LIN {X 0,Y 466.708,Z 598.278,A -85,B 0,C 180,E1 -7470,E2 -7470} C_VEL
LIN {X 0,Y 466.926,Z 594.295,A -85,B 0,C 180,E1 -7471.294,E2 -7471.294} C_VEL
LIN {X 0,Y 467.015,Z 589.345,A -85,B 0,C 180,E1 -7472.587,E2 -7472.587} C_VEL
LIN {X 0,Y 467.543,Z 582.26,A -85,B 0,C 180,E1 -7474.094,E2 -7474.094} C_VEL
LIN {X 0,Y 468.033,Z 573.535,A -85,B 0,C 180,E1 -7475.601,E2 -7475.601} C_VEL
LIN {X 0,Y 468.642,Z 564.398,A -85,B 0,C 180,E1 -7476.89,E2 -7476.89} C_VEL
LIN {X 0,Y 469.162,Z 555.335,A -85,B 0,C 180,E1 -7477.96,E2 -7477.96} C_VEL
LIN {X 0,Y 469.742,Z 543.987,A -85,B 0,C 180,E1 -7479.082,E2 -7479.082} C_VEL
LIN {X 0,Y 470.435,Z 532.566,A -85,B 0,C 180,E1 -7480.001,E2 -7480.001} C_VEL
LIN {X 0,Y 471.079,Z 519.327,A -85,B 0,C 180,E1 -7480.856,E2 -7480.856} C_VEL
LIN {X 0,Y 471.604,Z 506.561,A -85,B 0,C 180,E1 -7481.497,E2 -7481.497} C_VEL
LIN {X 0,Y 472.126,Z 492.888,A -85,B 0,C 180,E1 -7482.001,E2 -7482.001} C_VEL
LIN {X 0,Y 472.334,Z 478.929,A -85,B 0,C 180,E1 -7482.35,E2 -7482.35} C_VEL
LIN {X 0,Y 473.44,Z 363.18,A -85,B 0,C 180,E1 -7484.133,E2 -7484.133} C_VEL
LIN {X 0,Y 469.666,Z 345.085,A -85,B 0,C 180,E1 -7484.585,E2 -7484.585} C_VEL
LIN {X 0,Y 469.849,Z 337.166,A -85,B 0,C 180,E1 -7486.064,E2 -7486.064} C_VEL
LIN {X 0,Y 467.678,Z 325.858,A -85,B 0,C 180,E1 -7488.367,E2 -7488.367} C_VEL
LIN {X 0,Y 467.584,Z 325.868,A -85,B 0,C 180,E1 -7491.267,E2 -7491.267} C_VEL
LIN {X 0,Y 467.566,Z 325.871,A -85,B 0,C 180,E1 -7493.943,E2 -7493.943} C_VEL
LIN {X 0,Y 467.615,Z 325.859,A -85,B 0,C 180,E1 -7496.8,E2 -7496.8} C_VEL
LIN {X 0,Y 467.555,Z 325.871,A -85,B 0,C 180,E1 -7499.737,E2 -7499.737} C_VEL
LIN {X 0,Y 467.584,Z 325.862,A -85,B 0,C 180,E1 -7502.757,E2 -7502.757} C_VEL
LIN {X 0,Y 467.556,Z 325.867,A -85,B 0,C 180,E1 -7505.888,E2 -7505.888} C_VEL
LIN {X 0,Y 467.581,Z 325.865,A -85,B 0,C 180,E1 -7509.144,E2 -7509.144} C_VEL
LIN {X 0,Y 467.584,Z 325.861,A -85,B 0,C 180,E1 -7512.566,E2 -7512.566} C_VEL
LIN {X 0,Y 467.567,Z 325.866,A -85,B 0,C 180,E1 -7515.052,E2 -7515.052} C_VEL
LIN {X 0,Y 467.585,Z 325.866,A -85,B 0,C 180,E1 -7517.439,E2 -7517.439} C_VEL
LIN {X 0,Y 467.57,Z 325.866,A -85,B 0,C 180,E1 -7520.853,E2 -7520.853} C_VEL
LIN {X 0,Y 467.552,Z 325.866,A -85,B 0,C 180,E1 -7524.26,E2 -7524.26} C_VEL
LIN {X 0,Y 467.572,Z 325.868,A -85,B 0,C 180,E1 -7527.32,E2 -7527.32} C_VEL
LIN {X 0,Y 467.56,Z 325.867,A -85,B 0,C 180,E1 -7530.667,E2 -7530.667} C_VEL
LIN {X 0,Y 467.578,Z 325.863,A -85,B 0,C 180,E1 -7533.197,E2 -7533.197} C_VEL
LIN {X 0,Y 467.579,Z 325.864,A -85,B 0,C 180,E1 -7536.468,E2 -7536.468} C_VEL
LIN {X 0,Y 467.61,Z 325.85,A -85,B 0,C 180,E1 -7539.776,E2 -7539.776} C_VEL
LIN {X 0,Y 467.583,Z 325.863,A -85,B 0,C 180,E1 -7542.505,E2 -7542.505} C_VEL
LIN {X 0,Y 467.589,Z 325.86,A -85,B 0,C 180,E1 -7545.196,E2 -7545.196} C_VEL
LIN {X 0,Y 467.643,Z 325.845,A -85,B 0,C 180,E1 -7547.854,E2 -7547.854} C_VEL
LIN {X 0,Y 467.654,Z 325.854,A -85,B 0,C 180,E1 -7551.356,E2 -7551.356} C_VEL
LIN {X 0,Y 467.71,Z 325.843,A -85,B 0,C 180,E1 -7553.962,E2 -7553.962} C_VEL
LIN {X 0,Y 467.808,Z 325.831,A -85,B 0,C 180,E1 -7557.417,E2 -7557.417} C_VEL
LIN {X 0,Y 467.832,Z 325.832,A -85,B 0,C 180,E1 -7560,E2 -7560} C_VEL
LIN {X 0,Y 467.796,Z 325.835,A -85,B 0,C 180,E1 -7562.583,E2 -7562.583} C_VEL
LIN {X 0,Y 467.69,Z 325.851,A -85,B 0,C 180,E1 -7566.038,E2 -7566.038} C_VEL
LIN {X 0,Y 467.642,Z 325.853,A -85,B 0,C 180,E1 -7568.643,E2 -7568.643} C_VEL
LIN {X 0,Y 467.642,Z 325.859,A -85,B 0,C 180,E1 -7572.146,E2 -7572.146} C_VEL
LIN {X 0,Y 467.625,Z 325.853,A -85,B 0,C 180,E1 -7575.695,E2 -7575.695} C_VEL
LIN {X 0,Y 467.608,Z 325.858,A -85,B 0,C 180,E1 -7579.308,E2 -7579.308} C_VEL
LIN {X 0,Y 467.522,Z 325.87,A -85,B 0,C 180,E1 -7582.074,E2 -7582.074} C_VEL
LIN {X 0,Y 467.571,Z 325.861,A -85,B 0,C 180,E1 -7584.889,E2 -7584.889} C_VEL
LIN {X 0,Y 467.569,Z 325.866,A -85,B 0,C 180,E1 -7587.772,E2 -7587.772} C_VEL
LIN {X 0,Y 467.557,Z 325.863,A -85,B 0,C 180,E1 -7591.045,E2 -7591.045} C_VEL
LIN {X 0,Y 467.579,Z 325.865,A -85,B 0,C 180,E1 -7594.243,E2 -7594.243} C_VEL
LIN {X 0,Y 467.54,Z 325.868,A -85,B 0,C 180,E1 -7597.187,E2 -7597.187} C_VEL
LIN {X 0,Y 467.569,Z 325.862,A -85,B 0,C 180,E1 -7600.265,E2 -7600.265} C_VEL
LIN {X 0,Y 467.579,Z 325.861,A -85,B 0,C 180,E1 -7602.568,E2 -7602.568} C_VEL
LIN {X 0,Y 467.563,Z 325.865,A -85,B 0,C 180,E1 -7605.054,E2 -7605.054} C_VEL
LIN {X 0,Y 467.583,Z 325.867,A -85,B 0,C 180,E1 -7607.441,E2 -7607.441} C_VEL
LIN {X 0,Y 467.555,Z 325.869,A -85,B 0,C 180,E1 -7610.854,E2 -7610.854} C_VEL
LIN {X 0,Y 467.558,Z 325.869,A -85,B 0,C 180,E1 -7614.261,E2 -7614.261} C_VEL
LIN {X 0,Y 467.578,Z 325.87,A -85,B 0,C 180,E1 -7617.322,E2 -7617.322} C_VEL
LIN {X 0,Y 467.567,Z 325.867,A -85,B 0,C 180,E1 -7620.668,E2 -7620.668} C_VEL
LIN {X 0,Y 467.633,Z 325.91,A -85,B 0,C 180,E1 -7622.233,E2 -7622.233} C_VEL
LIN {X 0,Y 470.717,Z 340.455,A -85,B 0,C 180,E1 -7624.817,E2 -7624.817} C_VEL
LIN {X 0,Y 470.568,Z 347.177,A -85,B 0,C 180,E1 -7625.912,E2 -7625.912} C_VEL
LIN {X 0,Y 469.722,Z 364.766,A -85,B 0,C 180,E1 -7628.727,E2 -7628.727} C_VEL
LIN {X 0,Y 469.505,Z 369.198,A -85,B 0,C 180,E1 -7629.43,E2 -7629.43} C_VEL
LIN {X 0,Y 473.306,Z 391.122,A -85,B 0,C 180,E1 -7629.942,E2 -7629.942} C_VEL
LIN {X 0,Y 472.118,Z 506.928,A -85,B 0,C 180,E1 -7631.728,E2 -7631.728} C_VEL
LIN {X 0,Y 471.704,Z 521.762,A -85,B 0,C 180,E1 -7632.133,E2 -7632.133} C_VEL
LIN {X 0,Y 471.22,Z 535.785,A -85,B 0,C 180,E1 -7632.699,E2 -7632.699} C_VEL
LIN {X 0,Y 470.593,Z 549.174,A -85,B 0,C 180,E1 -7633.423,E2 -7633.423} C_VEL
LIN {X 0,Y 469.936,Z 561.542,A -85,B 0,C 180,E1 -7634.273,E2 -7634.273} C_VEL
LIN {X 0,Y 469.206,Z 573.078,A -85,B 0,C 180,E1 -7635.249,E2 -7635.249} C_VEL
LIN {X 0,Y 468.599,Z 583.669,A -85,B 0,C 180,E1 -7636.337,E2 -7636.337} C_VEL
LIN {X 0,Y 468.155,Z 593.288,A -85,B 0,C 180,E1 -7637.527,E2 -7637.527} C_VEL
LIN {X 0,Y 467.605,Z 602.864,A -85,B 0,C 180,E1 -7638.952,E2 -7638.952} C_VEL
LIN {X 0,Y 467.212,Z 611.173,A -85,B 0,C 180,E1 -7640.476,E2 -7640.476} C_VEL
LIN {X 0,Y 466.95,Z 616.974,A -85,B 0,C 180,E1 -7641.78,E2 -7641.78} C_VEL
LIN {X 0,Y 466.824,Z 621.733,A -85,B 0,C 180,E1 -7643.083,E2 -7643.083} C_VEL
LIN {X 0,Y 466.73,Z 626.661,A -85,B 0,C 180,E1 -7644.817,E2 -7644.817} C_VEL
LIN {X 0,Y 466.679,Z 630.086,A -85,B 0,C 180,E1 -7646.547,E2 -7646.547} C_VEL
LIN {X 0,Y 466.604,Z 632.111,A -85,B 0,C 180,E1 -7648.274,E2 -7648.274} C_VEL
LIN {X 0,Y 466.597,Z 632.785,A -85,B 0,C 180,E1 -7650,E2 -7650} C_VEL
LIN {X 0,Y 466.604,Z 632.119,A -85,B 0,C 180,E1 -7651.726,E2 -7651.726} C_VEL
LIN {X 0,Y 466.679,Z 630.104,A -85,B 0,C 180,E1 -7653.453,E2 -7653.453} C_VEL
LIN {X 0,Y 466.731,Z 626.692,A -85,B 0,C 180,E1 -7655.183,E2 -7655.183} C_VEL
LIN {X 0,Y 466.82,Z 621.782,A -85,B 0,C 180,E1 -7656.917,E2 -7656.917} C_VEL
LIN {X 0,Y 467.036,Z 615.237,A -85,B 0,C 180,E1 -7658.655,E2 -7658.655} C_VEL
LIN {X 0,Y 467.312,Z 607.962,A -85,B 0,C 180,E1 -7660.178,E2 -7660.178} C_VEL
LIN {X 0,Y 467.865,Z 598.973,A -85,B 0,C 180,E1 -7661.7,E2 -7661.7} C_VEL
LIN {X 0,Y 468.351,Z 589.551,A -85,B 0,C 180,E1 -7663.008,E2 -7663.008} C_VEL
LIN {X 0,Y 468.939,Z 579.134,A -85,B 0,C 180,E1 -7664.206,E2 -7664.206} C_VEL
LIN {X 0,Y 469.638,Z 567.661,A -85,B 0,C 180,E1 -7665.292,E2 -7665.292} C_VEL
LIN {X 0,Y 470.388,Z 554.968,A -85,B 0,C 180,E1 -7666.268,E2 -7666.268} C_VEL
LIN {X 0,Y 471.078,Z 542.255,A -85,B 0,C 180,E1 -7667.045,E2 -7667.045} C_VEL
LIN {X 0,Y 471.591,Z 528.59,A -85,B 0,C 180,E1 -7667.693,E2 -7667.693} C_VEL
LIN {X 0,Y 472.162,Z 513.986,A -85,B 0,C 180,E1 -7668.183,E2 -7668.183} C_VEL
LIN {X 0,Y 472.475,Z 499.718,A -85,B 0,C 180,E1 -7668.482,E2 -7668.482} C_VEL
LIN {X 0,Y 473.547,Z 391.005,A -85,B 0,C 180,E1 -7670.161,E2 -7670.161} C_VEL
LIN {X 0,Y 470.028,Z 371.07,A -85,B 0,C 180,E1 -7670.65,E2 -7670.65} C_VEL
LIN {X 0,Y 469.681,Z 368.925,A -85,B 0,C 180,E1 -7670.736,E2 -7670.736} C_VEL
LIN {X 0,Y 470.564,Z 351.6,A -85,B 0,C 180,E1 -7673.547,E2 -7673.547} C_VEL
LIN {X 0,Y 471.044,Z 341.783,A -85,B 0,C 180,E1 -7675.164,E2 -7675.164} C_VEL
LIN {X 0,Y 468.173,Z 328.175,A -85,B 0,C 180,E1 -7677.665,E2 -7677.665} C_VEL
LIN {X 0,Y 467.608,Z 325.863,A -85,B 0,C 180,E1 -7678.134,E2 -7678.134} C_VEL
LIN {X 0,Y 467.579,Z 325.867,A -85,B 0,C 180,E1 -7681.739,E2 -7681.739} C_VEL
LIN {X 0,Y 467.564,Z 325.868,A -85,B 0,C 180,E1 -7684.832,E2 -7684.832} C_VEL
LIN {X 0,Y 467.561,Z 325.862,A -85,B 0,C 180,E1 -7688.044,E2 -7688.044} C_VEL
LIN {X 0,Y 467.572,Z 325.859,A -85,B 0,C 180,E1 -7691.276,E2 -7691.276} C_VEL
LIN {X 0,Y 467.544,Z 325.866,A -85,B 0,C 180,E1 -7693.82,E2 -7693.82} C_VEL
LIN {X 0,Y 467.549,Z 325.871,A -85,B 0,C 180,E1 -7696.255,E2 -7696.255} C_VEL
LIN {X 0,Y 467.57,Z 325.865,A -85,B 0,C 180,E1 -7698.722,E2 -7698.722} C_VEL
LIN {X 0,Y 467.557,Z 325.872,A -85,B 0,C 180,E1 -7701.955,E2 -7701.955} C_VEL
LIN {X 0,Y 467.557,Z 325.863,A -85,B 0,C 180,E1 -7705.167,E2 -7705.167} C_VEL
LIN {X 0,Y 467.572,Z 325.861,A -85,B 0,C 180,E1 -7708.259,E2 -7708.259} C_VEL
LIN {X 0,Y 467.544,Z 325.859,A -85,B 0,C 180,E1 -7711.248,E2 -7711.248} C_VEL
LIN {X 0,Y 467.572,Z 325.866,A -85,B 0,C 180,E1 -7714.158,E2 -7714.158} C_VEL
LIN {X 0,Y 467.564,Z 325.864,A -85,B 0,C 180,E1 -7716.995,E2 -7716.995} C_VEL
LIN {X 0,Y 467.609,Z 325.861,A -85,B 0,C 180,E1 -7719.777,E2 -7719.777} C_VEL
LIN {X 0,Y 467.581,Z 325.862,A -85,B 0,C 180,E1 -7722.506,E2 -7722.506} C_VEL
LIN {X 0,Y 467.586,Z 325.862,A -85,B 0,C 180,E1 -7725.196,E2 -7725.196} C_VEL
LIN {X 0,Y 467.633,Z 325.856,A -85,B 0,C 180,E1 -7727.854,E2 -7727.854} C_VEL
LIN {X 0,Y 467.615,Z 325.864,A -85,B 0,C 180,E1 -7731.356,E2 -7731.356} C_VEL
LIN {X 0,Y 467.695,Z 325.85,A -85,B 0,C 180,E1 -7733.962,E2 -7733.962} C_VEL
LIN {X 0,Y 467.804,Z 325.836,A -85,B 0,C 180,E1 -7737.417,E2 -7737.417} C_VEL
LIN {X 0,Y 467.833,Z 325.832,A -85,B 0,C 180,E1 -7740,E2 -7740} C_VEL
LIN {X 0,Y 467.834,Z 325.827,A -85,B 0,C 180,E1 -7742.583,E2 -7742.583} C_VEL
LIN {X 0,Y 467.711,Z 325.845,A -85,B 0,C 180,E1 -7746.038,E2 -7746.038} C_VEL
LIN {X 0,Y 467.655,Z 325.852,A -85,B 0,C 180,E1 -7748.644,E2 -7748.644} C_VEL
LIN {X 0,Y 467.643,Z 325.849,A -85,B 0,C 180,E1 -7752.146,E2 -7752.146} C_VEL
LIN {X 0,Y 467.627,Z 325.855,A -85,B 0,C 180,E1 -7755.696,E2 -7755.696} C_VEL
LIN {X 0,Y 467.611,Z 325.861,A -85,B 0,C 180,E1 -7759.309,E2 -7759.309} C_VEL
LIN {X 0,Y 467.524,Z 325.869,A -85,B 0,C 180,E1 -7762.075,E2 -7762.075} C_VEL
LIN {X 0,Y 467.593,Z 325.864,A -85,B 0,C 180,E1 -7764.888,E2 -7764.888} C_VEL
LIN {X 0,Y 467.611,Z 325.856,A -85,B 0,C 180,E1 -7767.77,E2 -7767.77} C_VEL
LIN {X 0,Y 467.561,Z 325.866,A -85,B 0,C 180,E1 -7771.046,E2 -7771.046} C_VEL
LIN {X 0,Y 467.582,Z 325.864,A -85,B 0,C 180,E1 -7774.243,E2 -7774.243} C_VEL
LIN {X 0,Y 467.542,Z 325.866,A -85,B 0,C 180,E1 -7777.187,E2 -7777.187} C_VEL
LIN {X 0,Y 467.57,Z 325.867,A -85,B 0,C 180,E1 -7780.266,E2 -7780.266} C_VEL
LIN {X 0,Y 467.582,Z 325.867,A -85,B 0,C 180,E1 -7782.568,E2 -7782.568} C_VEL
LIN {X 0,Y 467.567,Z 325.867,A -85,B 0,C 180,E1 -7785.054,E2 -7785.054} C_VEL
LIN {X 0,Y 467.586,Z 325.863,A -85,B 0,C 180,E1 -7787.441,E2 -7787.441} C_VEL
LIN {X 0,Y 467.581,Z 325.866,A -85,B 0,C 180,E1 -7790.856,E2 -7790.856} C_VEL
LIN {X 0,Y 467.562,Z 325.871,A -85,B 0,C 180,E1 -7794.262,E2 -7794.262} C_VEL
LIN {X 0,Y 467.582,Z 325.867,A -85,B 0,C 180,E1 -7797.322,E2 -7797.322} C_VEL
LIN {X 0,Y 467.641,Z 326.019,A -85,B 0,C 180,E1 -7799.491,E2 -7799.491} C_VEL
LIN {X 0,Y 469.873,Z 336.684,A -85,B 0,C 180,E1 -7801.725,E2 -7801.725} C_VEL
LIN {X 0,Y 470.029,Z 341.316,A -85,B 0,C 180,E1 -7802.628,E2 -7802.628} C_VEL
LIN {X 0,Y 469.861,Z 345.182,A -85,B 0,C 180,E1 -7803.359,E2 -7803.359} C_VEL
LIN {X 0,Y 473.746,Z 362.881,A -85,B 0,C 180,E1 -7803.839,E2 -7803.839} C_VEL
LIN {X 0,Y 473.269,Z 414.35,A -85,B 0,C 180,E1 -7804.639,E2 -7804.639} C_VEL
LIN {X 0,Y 472.534,Z 420.197,A -85,B 0,C 180,E1 -7804.698,E2 -7804.698} C_VEL
LIN {X 0,Y 466.966,Z 439.231,A -85,B 0,C 180,E1 -7804.744,E2 -7804.744} C_VEL
LIN {X 0,Y 466.256,Z 445.077,A -85,B 0,C 180,E1 -7804.806,E2 -7804.806} C_VEL
LIN {X 0,Y 465.796,Z 482.934,A -85,B 0,C 180,E1 -7805.427,E2 -7805.427} C_VEL
LIN {X 0,Y 465.429,Z 496.712,A -85,B 0,C 180,E1 -7805.822,E2 -7805.822} C_VEL
LIN {X 0,Y 464.94,Z 510.311,A -85,B 0,C 180,E1 -7806.387,E2 -7806.387} C_VEL
LIN {X 0,Y 464.329,Z 522.416,A -85,B 0,C 180,E1 -7807.046,E2 -7807.046} C_VEL
LIN {X 0,Y 463.545,Z 535.599,A -85,B 0,C 180,E1 -7807.961,E2 -7807.961} C_VEL
LIN {X 0,Y 462.865,Z 547.324,A -85,B 0,C 180,E1 -7808.979,E2 -7808.979} C_VEL
LIN {X 0,Y 462.269,Z 557.036,A -85,B 0,C 180,E1 -7809.997,E2 -7809.997} C_VEL
LIN {X 0,Y 461.53,Z 567.777,A -85,B 0,C 180,E1 -7811.351,E2 -7811.351} C_VEL
LIN {X 0,Y 460.92,Z 576.598,A -85,B 0,C 180,E1 -7812.703,E2 -7812.703} C_VEL
LIN {X 0,Y 460.488,Z 584.531,A -85,B 0,C 180,E1 -7814.183,E2 -7814.183} C_VEL
LIN {X 0,Y 460.065,Z 591.723,A -85,B 0,C 180,E1 -7815.853,E2 -7815.853} C_VEL
LIN {X 0,Y 459.831,Z 597.64,A -85,B 0,C 180,E1 -7817.645,E2 -7817.645} C_VEL
LIN {X 0,Y 459.629,Z 601.949,A -85,B 0,C 180,E1 -7819.427,E2 -7819.427} C_VEL
LIN {X 0,Y 459.501,Z 604.787,A -85,B 0,C 180,E1 -7821.202,E2 -7821.202} C_VEL
LIN {X 0,Y 459.577,Z 606.244,A -85,B 0,C 180,E1 -7822.973,E2 -7822.973} C_VEL
LIN {X 0,Y 459.568,Z 606.371,A -85,B 0,C 180,E1 -7824.736,E2 -7824.736} C_VEL
LIN {X 0,Y 459.598,Z 605.178,A -85,B 0,C 180,E1 -7826.493,E2 -7826.493} C_VEL
LIN {X 0,Y 459.592,Z 602.646,A -85,B 0,C 180,E1 -7828.247,E2 -7828.247} C_VEL
LIN {X 0,Y 459.634,Z 598.697,A -85,B 0,C 180,E1 -7830,E2 -7830} C_VEL
LIN {X 0,Y 459.802,Z 593.221,A -85,B 0,C 180,E1 -7831.752,E2 -7831.752} C_VEL
LIN {X 0,Y 460.144,Z 588.034,A -85,B 0,C 180,E1 -7833.064,E2 -7833.064} C_VEL
LIN {X 0,Y 460.553,Z 580.575,A -85,B 0,C 180,E1 -7834.595,E2 -7834.595} C_VEL
LIN {X 0,Y 461.148,Z 572.81,A -85,B 0,C 180,E1 -7835.904,E2 -7835.904} C_VEL
LIN {X 0,Y 461.697,Z 563.475,A -85,B 0,C 180,E1 -7837.214,E2 -7837.214} C_VEL
LIN {X 0,Y 462.417,Z 552.137,A -85,B 0,C 180,E1 -7838.517,E2 -7838.517} C_VEL
LIN {X 0,Y 463.12,Z 540.502,A -85,B 0,C 180,E1 -7839.609,E2 -7839.609} C_VEL
LIN {X 0,Y 463.831,Z 527.615,A -85,B 0,C 180,E1 -7840.586,E2 -7840.586} C_VEL
LIN {X 0,Y 464.457,Z 514.954,A -85,B 0,C 180,E1 -7841.344,E2 -7841.344} C_VEL
LIN {X 0,Y 465.017,Z 500.663,A -85,B 0,C 180,E1 -7841.994,E2 -7841.994} C_VEL
LIN {X 0,Y 465.455,Z 487.156,A -85,B 0,C 180,E1 -7842.425,E2 -7842.425} C_VEL
LIN {X 0,Y 465.669,Z 472.206,A -85,B 0,C 180,E1 -7842.723,E2 -7842.723} C_VEL
LIN {X 0,Y 466.662,Z 363.736,A -85,B 0,C 180,E1 -7844.41,E2 -7844.41} C_VEL
LIN {X 0,Y 462.776,Z 345.273,A -85,B 0,C 180,E1 -7844.882,E2 -7844.882} C_VEL
LIN {X 0,Y 462.959,Z 339.043,A -85,B 0,C 180,E1 -7846.06,E2 -7846.06} C_VEL
LIN {X 0,Y 460.611,Z 326.738,A -85,B 0,C 180,E1 -7848.601,E2 -7848.601} C_VEL
LIN {X 0,Y 460.519,Z 326.748,A -85,B 0,C 180,E1 -7851.485,E2 -7851.485} C_VEL
LIN {X 0,Y 460.534,Z 326.744,A -85,B 0,C 180,E1 -7854.332,E2 -7854.332} C_VEL
LIN {X 0,Y 460.573,Z 326.738,A -85,B 0,C 180,E1 -7857.243,E2 -7857.243} C_VEL
LIN {X 0,Y 460.511,Z 326.745,A -85,B 0,C 180,E1 -7860.239,E2 -7860.239} C_VEL
LIN {X 0,Y 460.53,Z 326.744,A -85,B 0,C 180,E1 -7863.324,E2 -7863.324} C_VEL
LIN {X 0,Y 460.478,Z 326.746,A -85,B 0,C 180,E1 -7866.528,E2 -7866.528} C_VEL
LIN {X 0,Y 460.543,Z 326.74,A -85,B 0,C 180,E1 -7868.897,E2 -7868.897} C_VEL
LIN {X 0,Y 460.52,Z 326.742,A -85,B 0,C 180,E1 -7872.18,E2 -7872.18} C_VEL
LIN {X 0,Y 460.513,Z 326.747,A -85,B 0,C 180,E1 -7875.41,E2 -7875.41} C_VEL
LIN {X 0,Y 460.527,Z 326.738,A -85,B 0,C 180,E1 -7878.396,E2 -7878.396} C_VEL
LIN {X 0,Y 460.517,Z 326.747,A -85,B 0,C 180,E1 -7881.265,E2 -7881.265} C_VEL
LIN {X 0,Y 460.502,Z 326.745,A -85,B 0,C 180,E1 -7884.553,E2 -7884.553} C_VEL
LIN {X 0,Y 460.522,Z 326.743,A -85,B 0,C 180,E1 -7887.714,E2 -7887.714} C_VEL
LIN {X 0,Y 460.53,Z 326.743,A -85,B 0,C 180,E1 -7890.768,E2 -7890.768} C_VEL
LIN {X 0,Y 460.533,Z 326.738,A -85,B 0,C 180,E1 -7893.732,E2 -7893.732} C_VEL
LIN {X 0,Y 460.533,Z 326.743,A -85,B 0,C 180,E1 -7896.623,E2 -7896.623} C_VEL
LIN {X 0,Y 460.539,Z 326.732,A -85,B 0,C 180,E1 -7899.452,E2 -7899.452} C_VEL
LIN {X 0,Y 460.535,Z 326.739,A -85,B 0,C 180,E1 -7902.229,E2 -7902.229} C_VEL
LIN {X 0,Y 460.549,Z 326.74,A -85,B 0,C 180,E1 -7904.964,E2 -7904.964} C_VEL
LIN {X 0,Y 460.594,Z 326.728,A -85,B 0,C 180,E1 -7908.559,E2 -7908.559} C_VEL
LIN {X 0,Y 460.604,Z 326.733,A -85,B 0,C 180,E1 -7911.223,E2 -7911.223} C_VEL
LIN {X 0,Y 460.676,Z 326.718,A -85,B 0,C 180,E1 -7913.869,E2 -7913.869} C_VEL
LIN {X 0,Y 460.753,Z 326.71,A -85,B 0,C 180,E1 -7917.377,E2 -7917.377} C_VEL
LIN {X 0,Y 460.781,Z 326.711,A -85,B 0,C 180,E1 -7920,E2 -7920} C_VEL
LIN {X 0,Y 460.739,Z 326.713,A -85,B 0,C 180,E1 -7922.623,E2 -7922.623} C_VEL
LIN {X 0,Y 460.656,Z 326.728,A -85,B 0,C 180,E1 -7926.13,E2 -7926.13} C_VEL
LIN {X 0,Y 460.592,Z 326.729,A -85,B 0,C 180,E1 -7928.777,E2 -7928.777} C_VEL
LIN {X 0,Y 460.596,Z 326.74,A -85,B 0,C 180,E1 -7932.334,E2 -7932.334} C_VEL
LIN {X 0,Y 460.588,Z 326.732,A -85,B 0,C 180,E1 -7935.998,E2 -7935.998} C_VEL
LIN {X 0,Y 460.555,Z 326.738,A -85,B 0,C 180,E1 -7939.616,E2 -7939.616} C_VEL
LIN {X 0,Y 460.498,Z 326.747,A -85,B 0,C 180,E1 -7942.429,E2 -7942.429} C_VEL
LIN {X 0,Y 460.537,Z 326.742,A -85,B 0,C 180,E1 -7945.797,E2 -7945.797} C_VEL
LIN {X 0,Y 460.515,Z 326.746,A -85,B 0,C 180,E1 -7948.235,E2 -7948.235} C_VEL
LIN {X 0,Y 460.51,Z 326.742,A -85,B 0,C 180,E1 -7951.283,E2 -7951.283} C_VEL
LIN {X 0,Y 460.523,Z 326.742,A -85,B 0,C 180,E1 -7954.506,E2 -7954.506} C_VEL
LIN {X 0,Y 460.493,Z 326.749,A -85,B 0,C 180,E1 -7957.624,E2 -7957.624} C_VEL
LIN {X 0,Y 460.534,Z 326.738,A -85,B 0,C 180,E1 -7960.27,E2 -7960.27} C_VEL
LIN {X 0,Y 460.492,Z 326.747,A -85,B 0,C 180,E1 -7963.376,E2 -7963.376} C_VEL
LIN {X 0,Y 460.493,Z 326.745,A -85,B 0,C 180,E1 -7966.625,E2 -7966.625} C_VEL
LIN {X 0,Y 460.533,Z 326.748,A -85,B 0,C 180,E1 -7969.732,E2 -7969.732} C_VEL
LIN {X 0,Y 460.496,Z 326.748,A -85,B 0,C 180,E1 -7972.524,E2 -7972.524} C_VEL
LIN {X 0,Y 460.544,Z 326.747,A -85,B 0,C 180,E1 -7975.625,E2 -7975.625} C_VEL
LIN {X 0,Y 460.534,Z 326.744,A -85,B 0,C 180,E1 -7978.745,E2 -7978.745} C_VEL
LIN {X 0,Y 460.589,Z 326.754,A -85,B 0,C 180,E1 -7981.98,E2 -7981.98} C_VEL
LIN {X 0,Y 463.73,Z 341.536,A -85,B 0,C 180,E1 -7984.651,E2 -7984.651} C_VEL
LIN {X 0,Y 463.78,Z 346.746,A -85,B 0,C 180,E1 -7985.522,E2 -7985.522} C_VEL
LIN {X 0,Y 462.75,Z 365.849,A -85,B 0,C 180,E1 -7988.624,E2 -7988.624} C_VEL
LIN {X 0,Y 462.596,Z 368.996,A -85,B 0,C 180,E1 -7989.131,E2 -7989.131} C_VEL
LIN {X 0,Y 466.588,Z 391.857,A -85,B 0,C 180,E1 -7989.676,E2 -7989.676} C_VEL
LIN {X 0,Y 465.371,Z 505.737,A -85,B 0,C 180,E1 -7991.453,E2 -7991.453} C_VEL
LIN {X 0,Y 464.951,Z 520.254,A -85,B 0,C 180,E1 -7991.835,E2 -7991.835} C_VEL
LIN {X 0,Y 464.457,Z 534.11,A -85,B 0,C 180,E1 -7992.385,E2 -7992.385} C_VEL
LIN {X 0,Y 463.831,Z 547.475,A -85,B 0,C 180,E1 -7993.097,E2 -7993.097} C_VEL
LIN {X 0,Y 463.144,Z 559.678,A -85,B 0,C 180,E1 -7993.923,E2 -7993.923} C_VEL
LIN {X 0,Y 462.389,Z 571.512,A -85,B 0,C 180,E1 -7994.913,E2 -7994.913} C_VEL
LIN {X 0,Y 461.648,Z 583.319,A -85,B 0,C 180,E1 -7996.127,E2 -7996.127} C_VEL
LIN {X 0,Y 461.124,Z 593.701,A -85,B 0,C 180,E1 -7997.433,E2 -7997.433} C_VEL
LIN {X 0,Y 460.6,Z 602.57,A -85,B 0,C 180,E1 -7998.782,E2 -7998.782} C_VEL
LIN {X 0,Y 460.137,Z 610.903,A -85,B 0,C 180,E1 -8000.328,E2 -8000.328} C_VEL
LIN {X 0,Y 459.895,Z 616.716,A -85,B 0,C 180,E1 -8001.653,E2 -8001.653} C_VEL
LIN {X 0,Y 459.733,Z 621.49,A -85,B 0,C 180,E1 -8002.976,E2 -8002.976} C_VEL
LIN {X 0,Y 459.644,Z 626.43,A -85,B 0,C 180,E1 -8004.736,E2 -8004.736} C_VEL
LIN {X 0,Y 459.574,Z 629.865,A -85,B 0,C 180,E1 -8006.493,E2 -8006.493} C_VEL
LIN {X 0,Y 459.517,Z 631.899,A -85,B 0,C 180,E1 -8008.247,E2 -8008.247} C_VEL
LIN {X 0,Y 459.528,Z 632.583,A -85,B 0,C 180,E1 -8010,E2 -8010} C_VEL
LIN {X 0,Y 459.517,Z 631.927,A -85,B 0,C 180,E1 -8011.753,E2 -8011.753} C_VEL
LIN {X 0,Y 459.574,Z 629.921,A -85,B 0,C 180,E1 -8013.507,E2 -8013.507} C_VEL
LIN {X 0,Y 459.645,Z 626.518,A -85,B 0,C 180,E1 -8015.264,E2 -8015.264} C_VEL
LIN {X 0,Y 459.731,Z 621.621,A -85,B 0,C 180,E1 -8017.025,E2 -8017.025} C_VEL
LIN {X 0,Y 459.969,Z 615.091,A -85,B 0,C 180,E1 -8018.789,E2 -8018.789} C_VEL
LIN {X 0,Y 460.281,Z 607.833,A -85,B 0,C 180,E1 -8020.335,E2 -8020.335} C_VEL
LIN {X 0,Y 460.855,Z 598.874,A -85,B 0,C 180,E1 -8021.88,E2 -8021.88} C_VEL
LIN {X 0,Y 461.374,Z 589.482,A -85,B 0,C 180,E1 -8023.208,E2 -8023.208} C_VEL
LIN {X 0,Y 462.007,Z 579.098,A -85,B 0,C 180,E1 -8024.424,E2 -8024.424} C_VEL
LIN {X 0,Y 462.78,Z 567.67,A -85,B 0,C 180,E1 -8025.525,E2 -8025.525} C_VEL
LIN {X 0,Y 463.57,Z 555.031,A -85,B 0,C 180,E1 -8026.514,E2 -8026.514} C_VEL
LIN {X 0,Y 464.337,Z 541.823,A -85,B 0,C 180,E1 -8027.333,E2 -8027.333} C_VEL
LIN {X 0,Y 464.892,Z 527.674,A -85,B 0,C 180,E1 -8028.008,E2 -8028.008} C_VEL
LIN {X 0,Y 465.482,Z 513.412,A -85,B 0,C 180,E1 -8028.485,E2 -8028.485} C_VEL
LIN {X 0,Y 465.83,Z 499.018,A -85,B 0,C 180,E1 -8028.784,E2 -8028.784} C_VEL
LIN {X 0,Y 466.908,Z 391.619,A -85,B 0,C 180,E1 -8030.469,E2 -8030.469} C_VEL
LIN {X 0,Y 463.268,Z 371.301,A -85,B 0,C 180,E1 -8030.983,E2 -8030.983} C_VEL
LIN {X 0,Y 462.822,Z 368.792,A -85,B 0,C 180,E1 -8031.07,E2 -8031.07} C_VEL
LIN {X 0,Y 463.759,Z 351.567,A -85,B 0,C 180,E1 -8033.914,E2 -8033.914} C_VEL
LIN {X 0,Y 464.156,Z 343.163,A -85,B 0,C 180,E1 -8035.324,E2 -8035.324} C_VEL
LIN {X 0,Y 461.464,Z 330.448,A -85,B 0,C 180,E1 -8037.7,E2 -8037.7} C_VEL
LIN {X 0,Y 460.563,Z 326.74,A -85,B 0,C 180,E1 -8038.449,E2 -8038.449} C_VEL
LIN {X 0,Y 460.517,Z 326.747,A -85,B 0,C 180,E1 -8041.282,E2 -8041.282} C_VEL
LIN {X 0,Y 460.53,Z 326.747,A -85,B 0,C 180,E1 -8044.505,E2 -8044.505} C_VEL
LIN {X 0,Y 460.497,Z 326.739,A -85,B 0,C 180,E1 -8047.622,E2 -8047.622} C_VEL
LIN {X 0,Y 460.536,Z 326.736,A -85,B 0,C 180,E1 -8050.269,E2 -8050.269} C_VEL
LIN {X 0,Y 460.491,Z 326.742,A -85,B 0,C 180,E1 -8053.375,E2 -8053.375} C_VEL
LIN {X 0,Y 460.493,Z 326.746,A -85,B 0,C 180,E1 -8056.624,E2 -8056.624} C_VEL
LIN {X 0,Y 460.534,Z 326.742,A -85,B 0,C 180,E1 -8059.73,E2 -8059.73} C_VEL
LIN {X 0,Y 460.492,Z 326.749,A -85,B 0,C 180,E1 -8062.523,E2 -8062.523} C_VEL
LIN {X 0,Y 460.538,Z 326.74,A -85,B 0,C 180,E1 -8065.623,E2 -8065.623} C_VEL
LIN {X 0,Y 460.528,Z 326.734,A -85,B 0,C 180,E1 -8068.744,E2 -8068.744} C_VEL
LIN {X 0,Y 460.54,Z 326.742,A -85,B 0,C 180,E1 -8072.261,E2 -8072.261} C_VEL
LIN {X 0,Y 460.523,Z 326.739,A -85,B 0,C 180,E1 -8074.704,E2 -8074.704} C_VEL
LIN {X 0,Y 460.498,Z 326.749,A -85,B 0,C 180,E1 -8077.571,E2 -8077.571} C_VEL
LIN {X 0,Y 460.555,Z 326.738,A -85,B 0,C 180,E1 -8080.384,E2 -8080.384} C_VEL
LIN {X 0,Y 460.592,Z 326.734,A -85,B 0,C 180,E1 -8084.059,E2 -8084.059} C_VEL
LIN {X 0,Y 460.589,Z 326.735,A -85,B 0,C 180,E1 -8087.666,E2 -8087.666} C_VEL
LIN {X 0,Y 460.57,Z 326.74,A -85,B 0,C 180,E1 -8091.223,E2 -8091.223} C_VEL
LIN {X 0,Y 460.66,Z 326.727,A -85,B 0,C 180,E1 -8093.87,E2 -8093.87} C_VEL
LIN {X 0,Y 460.748,Z 326.715,A -85,B 0,C 180,E1 -8097.377,E2 -8097.377} C_VEL
LIN {X 0,Y 460.782,Z 326.711,A -85,B 0,C 180,E1 -8100,E2 -8100} C_VEL
LIN {X 0,Y 460.775,Z 326.707,A -85,B 0,C 180,E1 -8102.623,E2 -8102.623} C_VEL
LIN {X 0,Y 460.678,Z 326.721,A -85,B 0,C 180,E1 -8106.131,E2 -8106.131} C_VEL
LIN {X 0,Y 460.605,Z 326.731,A -85,B 0,C 180,E1 -8108.777,E2 -8108.777} C_VEL
LIN {X 0,Y 460.585,Z 326.729,A -85,B 0,C 180,E1 -8112.436,E2 -8112.436} C_VEL
LIN {X 0,Y 460.59,Z 326.73,A -85,B 0,C 180,E1 -8115.998,E2 -8115.998} C_VEL
LIN {X 0,Y 460.557,Z 326.737,A -85,B 0,C 180,E1 -8119.616,E2 -8119.616} C_VEL
LIN {X 0,Y 460.501,Z 326.746,A -85,B 0,C 180,E1 -8122.43,E2 -8122.43} C_VEL
LIN {X 0,Y 460.559,Z 326.737,A -85,B 0,C 180,E1 -8125.803,E2 -8125.803} C_VEL
LIN {X 0,Y 460.544,Z 326.738,A -85,B 0,C 180,E1 -8128.234,E2 -8128.234} C_VEL
LIN {X 0,Y 460.513,Z 326.742,A -85,B 0,C 180,E1 -8131.284,E2 -8131.284} C_VEL
LIN {X 0,Y 460.525,Z 326.744,A -85,B 0,C 180,E1 -8134.507,E2 -8134.507} C_VEL
LIN {X 0,Y 460.495,Z 326.743,A -85,B 0,C 180,E1 -8137.624,E2 -8137.624} C_VEL
LIN {X 0,Y 460.534,Z 326.743,A -85,B 0,C 180,E1 -8140.27,E2 -8140.27} C_VEL
LIN {X 0,Y 460.496,Z 326.746,A -85,B 0,C 180,E1 -8143.377,E2 -8143.377} C_VEL
LIN {X 0,Y 460.497,Z 326.75,A -85,B 0,C 180,E1 -8146.626,E2 -8146.626} C_VEL
LIN {X 0,Y 460.54,Z 326.743,A -85,B 0,C 180,E1 -8149.732,E2 -8149.732} C_VEL
LIN {X 0,Y 460.526,Z 326.747,A -85,B 0,C 180,E1 -8152.521,E2 -8152.521} C_VEL
LIN {X 0,Y 460.548,Z 326.738,A -85,B 0,C 180,E1 -8155.625,E2 -8155.625} C_VEL
LIN {X 0,Y 460.533,Z 326.746,A -85,B 0,C 180,E1 -8159.001,E2 -8159.001} C_VEL
LIN {X 0,Y 460.566,Z 326.884,A -85,B 0,C 180,E1 -8159.194,E2 -8159.194} C_VEL
LIN {X 0,Y 462.795,Z 337.043,A -85,B 0,C 180,E1 -8161.368,E2 -8161.368} C_VEL
LIN {X 0,Y 463.216,Z 341.101,A -85,B 0,C 180,E1 -8162.191,E2 -8162.191} C_VEL
LIN {X 0,Y 463.074,Z 345.617,A -85,B 0,C 180,E1 -8163.025,E2 -8163.025} C_VEL
LIN {X 0,Y 467.174,Z 363.934,A -85,B 0,C 180,E1 -8163.534,E2 -8163.534} C_VEL
LIN {X 0,Y 466.256,Z 445.077,A -85,B 0,C 180,E1 -8164.806,E2 -8164.806} C_VEL
LIN {X 0,Y 465.545,Z 450.926,A -85,B 0,C 180,E1 -8164.865,E2 -8164.865} C_VEL
LIN {X 0,Y 460,Z 469.969,A -85,B 0,C 180,E1 -8164.909,E2 -8164.909} C_VEL
LIN {X 0,Y 459.293,Z 475.806,A -85,B 0,C 180,E1 -8164.98,E2 -8164.98} C_VEL
LIN {X 0,Y 458.967,Z 490.229,A -85,B 0,C 180,E1 -8165.308,E2 -8165.308} C_VEL
LIN {X 0,Y 458.531,Z 503.884,A -85,B 0,C 180,E1 -8165.796,E2 -8165.796} C_VEL
LIN {X 0,Y 457.821,Z 517.781,A -85,B 0,C 180,E1 -8166.477,E2 -8166.477} C_VEL
LIN {X 0,Y 457.219,Z 530.012,A -85,B 0,C 180,E1 -8167.262,E2 -8167.262} C_VEL
LIN {X 0,Y 456.385,Z 541.767,A -85,B 0,C 180,E1 -8168.192,E2 -8168.192} C_VEL
LIN {X 0,Y 455.555,Z 553.505,A -85,B 0,C 180,E1 -8169.336,E2 -8169.336} C_VEL
LIN {X 0,Y 454.896,Z 564.045,A -85,B 0,C 180,E1 -8170.594,E2 -8170.594} C_VEL
LIN {X 0,Y 454.204,Z 573.598,A -85,B 0,C 180,E1 -8171.974,E2 -8171.974} C_VEL
LIN {X 0,Y 453.686,Z 581.449,A -85,B 0,C 180,E1 -8173.347,E2 -8173.347} C_VEL
LIN {X 0,Y 453.276,Z 587.934,A -85,B 0,C 180,E1 -8174.718,E2 -8174.718} C_VEL
LIN {X 0,Y 452.943,Z 593.275,A -85,B 0,C 180,E1 -8176.084,E2 -8176.084} C_VEL
LIN {X 0,Y 452.78,Z 597.63,A -85,B 0,C 180,E1 -8177.449,E2 -8177.449} C_VEL
LIN {X 0,Y 452.562,Z 601.998,A -85,B 0,C 180,E1 -8179.26,E2 -8179.26} C_VEL
LIN {X 0,Y 452.42,Z 604.893,A -85,B 0,C 180,E1 -8181.064,E2 -8181.064} C_VEL
LIN {X 0,Y 452.474,Z 606.405,A -85,B 0,C 180,E1 -8182.862,E2 -8182.862} C_VEL
LIN {X 0,Y 452.483,Z 606.586,A -85,B 0,C 180,E1 -8184.653,E2 -8184.653} C_VEL
LIN {X 0,Y 452.493,Z 605.448,A -85,B 0,C 180,E1 -8186.438,E2 -8186.438} C_VEL
LIN {X 0,Y 452.503,Z 602.98,A -85,B 0,C 180,E1 -8188.22,E2 -8188.22} C_VEL
LIN {X 0,Y 452.562,Z 599.107,A -85,B 0,C 180,E1 -8190,E2 -8190} C_VEL
LIN {X 0,Y 452.736,Z 593.692,A -85,B 0,C 180,E1 -8191.779,E2 -8191.779} C_VEL
LIN {X 0,Y 453.075,Z 588.563,A -85,B 0,C 180,E1 -8193.112,E2 -8193.112} C_VEL
LIN {X 0,Y 453.527,Z 581.182,A -85,B 0,C 180,E1 -8194.666,E2 -8194.666} C_VEL
LIN {X 0,Y 454.139,Z 573.491,A -85,B 0,C 180,E1 -8195.996,E2 -8195.996} C_VEL
LIN {X 0,Y 454.71,Z 564.256,A -85,B 0,C 180,E1 -8197.326,E2 -8197.326} C_VEL
LIN {X 0,Y 455.466,Z 553.035,A -85,B 0,C 180,E1 -8198.648,E2 -8198.648} C_VEL
LIN {X 0,Y 456.105,Z 542.787,A -85,B 0,C 180,E1 -8199.648,E2 -8199.648} C_VEL
LIN {X 0,Y 456.862,Z 530.385,A -85,B 0,C 180,E1 -8200.637,E2 -8200.637} C_VEL
LIN {X 0,Y 457.51,Z 518.377,A -85,B 0,C 180,E1 -8201.407,E2 -8201.407} C_VEL
LIN {X 0,Y 458.054,Z 505.19,A -85,B 0,C 180,E1 -8202.066,E2 -8202.066} C_VEL
LIN {X 0,Y 458.602,Z 490.789,A -85,B 0,C 180,E1 -8202.585,E2 -8202.585} C_VEL
LIN {X 0,Y 458.864,Z 476.659,A -85,B 0,C 180,E1 -8202.915,E2 -8202.915} C_VEL
LIN {X 0,Y 459.961,Z 364.757,A -85,B 0,C 180,E1 -8204.683,E2 -8204.683} C_VEL
LIN {X 0,Y 455.899,Z 345.429,A -85,B 0,C 180,E1 -8205.192,E2 -8205.192} C_VEL
LIN {X 0,Y 456.046,Z 340.674,A -85,B 0,C 180,E1 -8206.104,E2 -8206.104} C_VEL
LIN {X 0,Y 453.873,Z 329.044,A -85,B 0,C 180,E1 -8208.507,E2 -8208.507} C_VEL
LIN {X 0,Y 453.552,Z 327.617,A -85,B 0,C 180,E1 -8208.84,E2 -8208.84} C_VEL
LIN {X 0,Y 453.48,Z 327.626,A -85,B 0,C 180,E1 -8211.835,E2 -8211.835} C_VEL
LIN {X 0,Y 453.503,Z 327.618,A -85,B 0,C 180,E1 -8214.734,E2 -8214.734} C_VEL
LIN {X 0,Y 453.534,Z 327.616,A -85,B 0,C 180,E1 -8217.959,E2 -8217.959} C_VEL
LIN {X 0,Y 453.467,Z 327.626,A -85,B 0,C 180,E1 -8221.524,E2 -8221.524} C_VEL
LIN {X 0,Y 453.489,Z 327.617,A -85,B 0,C 180,E1 -8224.776,E2 -8224.776} C_VEL
LIN {X 0,Y 453.472,Z 327.62,A -85,B 0,C 180,E1 -8228.31,E2 -8228.31} C_VEL
LIN {X 0,Y 453.492,Z 327.607,A -85,B 0,C 180,E1 -8230.608,E2 -8230.608} C_VEL
LIN {X 0,Y 453.453,Z 327.627,A -85,B 0,C 180,E1 -8233.243,E2 -8233.243} C_VEL
LIN {X 0,Y 453.462,Z 327.625,A -85,B 0,C 180,E1 -8235.778,E2 -8235.778} C_VEL
LIN {X 0,Y 453.474,Z 327.616,A -85,B 0,C 180,E1 -8238.208,E2 -8238.208} C_VEL
LIN {X 0,Y 453.486,Z 327.62,A -85,B 0,C 180,E1 -8240.793,E2 -8240.793} C_VEL
LIN {X 0,Y 453.447,Z 327.624,A -85,B 0,C 180,E1 -8243.916,E2 -8243.916} C_VEL
LIN {X 0,Y 453.471,Z 327.622,A -85,B 0,C 180,E1 -8247.15,E2 -8247.15} C_VEL
LIN {X 0,Y 453.466,Z 327.62,A -85,B 0,C 180,E1 -8250.267,E2 -8250.267} C_VEL
LIN {X 0,Y 453.523,Z 327.606,A -85,B 0,C 180,E1 -8252.296,E2 -8252.296} C_VEL
LIN {X 0,Y 453.483,Z 327.623,A -85,B 0,C 180,E1 -8255.263,E2 -8255.263} C_VEL
LIN {X 0,Y 453.47,Z 327.618,A -85,B 0,C 180,E1 -8258.414,E2 -8258.414} C_VEL
LIN {X 0,Y 453.512,Z 327.615,A -85,B 0,C 180,E1 -8261.008,E2 -8261.008} C_VEL
LIN {X 0,Y 453.558,Z 327.609,A -85,B 0,C 180,E1 -8263.879,E2 -8263.879} C_VEL
LIN {X 0,Y 453.553,Z 327.6,A -85,B 0,C 180,E1 -8267.47,E2 -8267.47} C_VEL
LIN {X 0,Y 453.57,Z 327.611,A -85,B 0,C 180,E1 -8271.086,E2 -8271.086} C_VEL
LIN {X 0,Y 453.644,Z 327.594,A -85,B 0,C 180,E1 -8273.774,E2 -8273.774} C_VEL
LIN {X 0,Y 453.7,Z 327.589,A -85,B 0,C 180,E1 -8277.336,E2 -8277.336} C_VEL
LIN {X 0,Y 453.732,Z 327.589,A -85,B 0,C 180,E1 -8280,E2 -8280} C_VEL
LIN {X 0,Y 453.686,Z 327.591,A -85,B 0,C 180,E1 -8282.663,E2 -8282.663} C_VEL
LIN {X 0,Y 453.623,Z 327.605,A -85,B 0,C 180,E1 -8286.226,E2 -8286.226} C_VEL
LIN {X 0,Y 453.559,Z 327.604,A -85,B 0,C 180,E1 -8288.914,E2 -8288.914} C_VEL
LIN {X 0,Y 453.552,Z 327.615,A -85,B 0,C 180,E1 -8292.529,E2 -8292.529} C_VEL
LIN {X 0,Y 453.532,Z 327.612,A -85,B 0,C 180,E1 -8296.196,E2 -8296.196} C_VEL
LIN {X 0,Y 453.505,Z 327.615,A -85,B 0,C 180,E1 -8299.039,E2 -8299.039} C_VEL
LIN {X 0,Y 453.465,Z 327.617,A -85,B 0,C 180,E1 -8301.837,E2 -8301.837} C_VEL
LIN {X 0,Y 453.488,Z 327.616,A -85,B 0,C 180,E1 -8304.736,E2 -8304.736} C_VEL
LIN {X 0,Y 453.495,Z 327.622,A -85,B 0,C 180,E1 -8307.954,E2 -8307.954} C_VEL
LIN {X 0,Y 453.465,Z 327.619,A -85,B 0,C 180,E1 -8310.76,E2 -8310.76} C_VEL
LIN {X 0,Y 453.468,Z 327.624,A -85,B 0,C 180,E1 -8313.913,E2 -8313.913} C_VEL
LIN {X 0,Y 453.444,Z 327.624,A -85,B 0,C 180,E1 -8317.19,E2 -8317.19} C_VEL
LIN {X 0,Y 453.508,Z 327.619,A -85,B 0,C 180,E1 -8319.448,E2 -8319.448} C_VEL
LIN {X 0,Y 453.456,Z 327.621,A -85,B 0,C 180,E1 -8322.996,E2 -8322.996} C_VEL
LIN {X 0,Y 453.459,Z 327.628,A -85,B 0,C 180,E1 -8325.78,E2 -8325.78} C_VEL
LIN {X 0,Y 453.473,Z 327.622,A -85,B 0,C 180,E1 -8328.21,E2 -8328.21} C_VEL
LIN {X 0,Y 453.482,Z 327.622,A -85,B 0,C 180,E1 -8330.795,E2 -8330.795} C_VEL
LIN {X 0,Y 453.452,Z 327.629,A -85,B 0,C 180,E1 -8333.918,E2 -8333.918} C_VEL
LIN {X 0,Y 453.479,Z 327.626,A -85,B 0,C 180,E1 -8337.152,E2 -8337.152} C_VEL
LIN {X 0,Y 453.472,Z 327.622,A -85,B 0,C 180,E1 -8340.269,E2 -8340.269} C_VEL
LIN {X 0,Y 453.558,Z 327.67,A -85,B 0,C 180,E1 -8341.732,E2 -8341.732} C_VEL
LIN {X 0,Y 456.724,Z 342.607,A -85,B 0,C 180,E1 -8344.479,E2 -8344.479} C_VEL
LIN {X 0,Y 456.936,Z 346.546,A -85,B 0,C 180,E1 -8345.157,E2 -8345.157} C_VEL
LIN {X 0,Y 455.875,Z 365.497,A -85,B 0,C 180,E1 -8348.285,E2 -8348.285} C_VEL
LIN {X 0,Y 455.704,Z 368.824,A -85,B 0,C 180,E1 -8348.831,E2 -8348.831} C_VEL
LIN {X 0,Y 459.849,Z 393.633,A -85,B 0,C 180,E1 -8349.421,E2 -8349.421} C_VEL
LIN {X 0,Y 458.605,Z 505.894,A -85,B 0,C 180,E1 -8351.199,E2 -8351.199} C_VEL
LIN {X 0,Y 458.144,Z 520.243,A -85,B 0,C 180,E1 -8351.585,E2 -8351.585} C_VEL
LIN {X 0,Y 457.613,Z 534.505,A -85,B 0,C 180,E1 -8352.164,E2 -8352.164} C_VEL
LIN {X 0,Y 456.976,Z 547.262,A -85,B 0,C 180,E1 -8352.856,E2 -8352.856} C_VEL
LIN {X 0,Y 456.191,Z 560.652,A -85,B 0,C 180,E1 -8353.786,E2 -8353.786} C_VEL
LIN {X 0,Y 455.403,Z 572.284,A -85,B 0,C 180,E1 -8354.791,E2 -8354.791} C_VEL
LIN {X 0,Y 454.674,Z 582.946,A -85,B 0,C 180,E1 -8355.91,E2 -8355.91} C_VEL
LIN {X 0,Y 454.105,Z 592.867,A -85,B 0,C 180,E1 -8357.168,E2 -8357.168} C_VEL
LIN {X 0,Y 453.59,Z 602.259,A -85,B 0,C 180,E1 -8358.607,E2 -8358.607} C_VEL
LIN {X 0,Y 453.071,Z 610.619,A -85,B 0,C 180,E1 -8360.176,E2 -8360.176} C_VEL
LIN {X 0,Y 452.822,Z 616.445,A -85,B 0,C 180,E1 -8361.521,E2 -8361.521} C_VEL
LIN {X 0,Y 452.656,Z 621.236,A -85,B 0,C 180,E1 -8362.865,E2 -8362.865} C_VEL
LIN {X 0,Y 452.559,Z 626.192,A -85,B 0,C 180,E1 -8364.654,E2 -8364.654} C_VEL
LIN {X 0,Y 452.471,Z 629.639,A -85,B 0,C 180,E1 -8366.438,E2 -8366.438} C_VEL
LIN {X 0,Y 452.504,Z 630.834,A -85,B 0,C 180,E1 -8367.329,E2 -8367.329} C_VEL
LIN {X 0,Y 452.426,Z 632.201,A -85,B 0,C 180,E1 -8369.11,E2 -8369.11} C_VEL
LIN {X 0,Y 452.426,Z 632.226,A -85,B 0,C 180,E1 -8370.89,E2 -8370.89} C_VEL
LIN {X 0,Y 452.504,Z 630.913,A -85,B 0,C 180,E1 -8372.671,E2 -8372.671} C_VEL
LIN {X 0,Y 452.472,Z 628.227,A -85,B 0,C 180,E1 -8374.454,E2 -8374.454} C_VEL
LIN {X 0,Y 452.602,Z 624.107,A -85,B 0,C 180,E1 -8376.24,E2 -8376.24} C_VEL
LIN {X 0,Y 452.742,Z 618.429,A -85,B 0,C 180,E1 -8378.031,E2 -8378.031} C_VEL
LIN {X 0,Y 453.065,Z 612.038,A -85,B 0,C 180,E1 -8379.599,E2 -8379.599} C_VEL
LIN {X 0,Y 453.543,Z 604.106,A -85,B 0,C 180,E1 -8381.168,E2 -8381.168} C_VEL
LIN {X 0,Y 454.058,Z 594.986,A -85,B 0,C 180,E1 -8382.643,E2 -8382.643} C_VEL
LIN {X 0,Y 454.658,Z 585.867,A -85,B 0,C 180,E1 -8383.862,E2 -8383.862} C_VEL
LIN {X 0,Y 455.385,Z 574.811,A -85,B 0,C 180,E1 -8385.095,E2 -8385.095} C_VEL
LIN {X 0,Y 456.315,Z 562.472,A -85,B 0,C 180,E1 -8386.209,E2 -8386.209} C_VEL
LIN {X 0,Y 457.114,Z 549.348,A -85,B 0,C 180,E1 -8387.159,E2 -8387.159} C_VEL
LIN {X 0,Y 457.889,Z 535.581,A -85,B 0,C 180,E1 -8387.934,E2 -8387.934} C_VEL
LIN {X 0,Y 458.43,Z 522.499,A -85,B 0,C 180,E1 -8388.49,E2 -8388.49} C_VEL
LIN {X 0,Y 458.963,Z 508.487,A -85,B 0,C 180,E1 -8388.902,E2 -8388.902} C_VEL
LIN {X 0,Y 459.353,Z 482.477,A -85,B 0,C 180,E1 -8389.349,E2 -8389.349} C_VEL
LIN {X 0,Y 460.333,Z 392.723,A -85,B 0,C 180,E1 -8390.778,E2 -8390.778} C_VEL
LIN {X 0,Y 456.823,Z 373.013,A -85,B 0,C 180,E1 -8391.286,E2 -8391.286} C_VEL
LIN {X 0,Y 455.995,Z 368.691,A -85,B 0,C 180,E1 -8391.411,E2 -8391.411} C_VEL
LIN {X 0,Y 457.009,Z 351.543,A -85,B 0,C 180,E1 -8394.29,E2 -8394.29} C_VEL
LIN {X 0,Y 457.27,Z 344.55,A -85,B 0,C 180,E1 -8395.489,E2 -8395.489} C_VEL
LIN {X 0,Y 454.482,Z 331.733,A -85,B 0,C 180,E1 -8397.935,E2 -8397.935} C_VEL
LIN {X 0,Y 453.5,Z 327.622,A -85,B 0,C 180,E1 -8398.775,E2 -8398.775} C_VEL
LIN {X 0,Y 453.461,Z 327.626,A -85,B 0,C 180,E1 -8401.799,E2 -8401.799} C_VEL
LIN {X 0,Y 453.478,Z 327.622,A -85,B 0,C 180,E1 -8404.988,E2 -8404.988} C_VEL
LIN {X 0,Y 453.46,Z 327.622,A -85,B 0,C 180,E1 -8408.311,E2 -8408.311} C_VEL
LIN {X 0,Y 453.488,Z 327.614,A -85,B 0,C 180,E1 -8410.608,E2 -8410.608} C_VEL
LIN {X 0,Y 453.447,Z 327.619,A -85,B 0,C 180,E1 -8413.243,E2 -8413.243} C_VEL
LIN {X 0,Y 453.459,Z 327.619,A -85,B 0,C 180,E1 -8415.778,E2 -8415.778} C_VEL
LIN {X 0,Y 453.472,Z 327.625,A -85,B 0,C 180,E1 -8418.209,E2 -8418.209} C_VEL
LIN {X 0,Y 453.486,Z 327.62,A -85,B 0,C 180,E1 -8420.793,E2 -8420.793} C_VEL
LIN {X 0,Y 453.447,Z 327.628,A -85,B 0,C 180,E1 -8423.917,E2 -8423.917} C_VEL
LIN {X 0,Y 453.473,Z 327.62,A -85,B 0,C 180,E1 -8427.151,E2 -8427.151} C_VEL
LIN {X 0,Y 453.456,Z 327.612,A -85,B 0,C 180,E1 -8430.267,E2 -8430.267} C_VEL
LIN {X 0,Y 453.46,Z 327.622,A -85,B 0,C 180,E1 -8433.291,E2 -8433.291} C_VEL
LIN {X 0,Y 453.483,Z 327.621,A -85,B 0,C 180,E1 -8436.238,E2 -8436.238} C_VEL
LIN {X 0,Y 453.47,Z 327.619,A -85,B 0,C 180,E1 -8439.117,E2 -8439.117} C_VEL
LIN {X 0,Y 453.489,Z 327.622,A -85,B 0,C 180,E1 -8441.944,E2 -8441.944} C_VEL
LIN {X 0,Y 453.524,Z 327.611,A -85,B 0,C 180,E1 -8444.726,E2 -8444.726} C_VEL
LIN {X 0,Y 453.529,Z 327.608,A -85,B 0,C 180,E1 -8448.378,E2 -8448.378} C_VEL
LIN {X 0,Y 453.541,Z 327.614,A -85,B 0,C 180,E1 -8451.086,E2 -8451.086} C_VEL
LIN {X 0,Y 453.626,Z 327.604,A -85,B 0,C 180,E1 -8453.774,E2 -8453.774} C_VEL
LIN {X 0,Y 453.695,Z 327.594,A -85,B 0,C 180,E1 -8457.337,E2 -8457.337} C_VEL
LIN {X 0,Y 453.733,Z 327.589,A -85,B 0,C 180,E1 -8460,E2 -8460} C_VEL
LIN {X 0,Y 453.719,Z 327.586,A -85,B 0,C 180,E1 -8462.664,E2 -8462.664} C_VEL
LIN {X 0,Y 453.646,Z 327.597,A -85,B 0,C 180,E1 -8466.226,E2 -8466.226} C_VEL
LIN {X 0,Y 453.571,Z 327.609,A -85,B 0,C 180,E1 -8468.914,E2 -8468.914} C_VEL
LIN {X 0,Y 453.553,Z 327.605,A -85,B 0,C 180,E1 -8472.53,E2 -8472.53} C_VEL
LIN {X 0,Y 453.534,Z 327.609,A -85,B 0,C 180,E1 -8476.197,E2 -8476.197} C_VEL
LIN {X 0,Y 453.507,Z 327.621,A -85,B 0,C 180,E1 -8479.04,E2 -8479.04} C_VEL
LIN {X 0,Y 453.467,Z 327.62,A -85,B 0,C 180,E1 -8481.837,E2 -8481.837} C_VEL
LIN {X 0,Y 453.504,Z 327.618,A -85,B 0,C 180,E1 -8484.735,E2 -8484.735} C_VEL
LIN {X 0,Y 453.524,Z 327.611,A -85,B 0,C 180,E1 -8487.96,E2 -8487.96} C_VEL
LIN {X 0,Y 453.458,Z 327.619,A -85,B 0,C 180,E1 -8491.526,E2 -8491.526} C_VEL
LIN {X 0,Y 453.481,Z 327.622,A -85,B 0,C 180,E1 -8494.778,E2 -8494.778} C_VEL
LIN {X 0,Y 453.455,Z 327.624,A -85,B 0,C 180,E1 -8498.313,E2 -8498.313} C_VEL
LIN {X 0,Y 453.489,Z 327.622,A -85,B 0,C 180,E1 -8500.61,E2 -8500.61} C_VEL
LIN {X 0,Y 453.452,Z 327.624,A -85,B 0,C 180,E1 -8503.245,E2 -8503.245} C_VEL
LIN {X 0,Y 453.463,Z 327.624,A -85,B 0,C 180,E1 -8505.78,E2 -8505.78} C_VEL
LIN {X 0,Y 453.477,Z 327.626,A -85,B 0,C 180,E1 -8508.21,E2 -8508.21} C_VEL
LIN {X 0,Y 453.514,Z 327.619,A -85,B 0,C 180,E1 -8510.791,E2 -8510.791} C_VEL
LIN {X 0,Y 453.456,Z 327.627,A -85,B 0,C 180,E1 -8513.918,E2 -8513.918} C_VEL
LIN {X 0,Y 453.483,Z 327.623,A -85,B 0,C 180,E1 -8517.152,E2 -8517.152} C_VEL
LIN {X 0,Y 453.513,Z 327.696,A -85,B 0,C 180,E1 -8518.876,E2 -8518.876} C_VEL
LIN {X 0,Y 456.087,Z 339.625,A -85,B 0,C 180,E1 -8521.466,E2 -8521.466} C_VEL
LIN {X 0,Y 456.311,Z 343.411,A -85,B 0,C 180,E1 -8522.232,E2 -8522.232} C_VEL
LIN {X 0,Y 456.242,Z 345.823,A -85,B 0,C 180,E1 -8522.667,E2 -8522.667} C_VEL
LIN {X 0,Y 460.64,Z 365.49,A -85,B 0,C 180,E1 -8523.227,E2 -8523.227} C_VEL
LIN {X 0,Y 459.293,Z 475.806,A -85,B 0,C 180,E1 -8524.98,E2 -8524.98} C_VEL
LIN {X 0,Y 458.545,Z 481.628,A -85,B 0,C 180,E1 -8525.058,E2 -8525.058} C_VEL
LIN {X 0,Y 455.612,Z 491.058,A -85,B 0,C 180,E1 -8525.176,E2 -8525.176} C_VEL
LIN {X 0,Y 452.626,Z 500.411,A -85,B 0,C 180,E1 -8525.369,E2 -8525.369} C_VEL
LIN {X 0,Y 451.774,Z 505.959,A -85,B 0,C 180,E1 -8525.573,E2 -8525.573} C_VEL
LIN {X 0,Y 451.084,Z 518.947,A -85,B 0,C 180,E1 -8526.238,E2 -8526.238} C_VEL
LIN {X 0,Y 450.424,Z 531.087,A -85,B 0,C 180,E1 -8527.041,E2 -8527.041} C_VEL
LIN {X 0,Y 449.561,Z 542.453,A -85,B 0,C 180,E1 -8527.964,E2 -8527.964} C_VEL
LIN {X 0,Y 448.675,Z 554.102,A -85,B 0,C 180,E1 -8529.124,E2 -8529.124} C_VEL
LIN {X 0,Y 447.973,Z 564.585,A -85,B 0,C 180,E1 -8530.403,E2 -8530.403} C_VEL
LIN {X 0,Y 447.18,Z 574.736,A -85,B 0,C 180,E1 -8531.917,E2 -8531.917} C_VEL
LIN {X 0,Y 446.567,Z 583.556,A -85,B 0,C 180,E1 -8533.544,E2 -8533.544} C_VEL
LIN {X 0,Y 446.156,Z 589.73,A -85,B 0,C 180,E1 -8534.936,E2 -8534.936} C_VEL
LIN {X 0,Y 445.853,Z 594.819,A -85,B 0,C 180,E1 -8536.324,E2 -8536.324} C_VEL
LIN {X 0,Y 445.627,Z 600.032,A -85,B 0,C 180,E1 -8538.169,E2 -8538.169} C_VEL
LIN {X 0,Y 445.363,Z 603.705,A -85,B 0,C 180,E1 -8540.004,E2 -8540.004} C_VEL
LIN {X 0,Y 445.347,Z 605.953,A -85,B 0,C 180,E1 -8541.835,E2 -8541.835} C_VEL
LIN {X 0,Y 445.435,Z 606.86,A -85,B 0,C 180,E1 -8543.727,E2 -8543.727} C_VEL
LIN {X 0,Y 445.362,Z 606.424,A -85,B 0,C 180,E1 -8545.475,E2 -8545.475} C_VEL
LIN {X 0,Y 445.447,Z 604.675,A -85,B 0,C 180,E1 -8547.287,E2 -8547.287} C_VEL
LIN {X 0,Y 445.471,Z 601.579,A -85,B 0,C 180,E1 -8549.096,E2 -8549.096} C_VEL
LIN {X 0,Y 445.556,Z 597.032,A -85,B 0,C 180,E1 -8550.904,E2 -8550.904} C_VEL
LIN {X 0,Y 445.849,Z 590.856,A -85,B 0,C 180,E1 -8552.71,E2 -8552.71} C_VEL
LIN {X 0,Y 446.376,Z 583.978,A -85,B 0,C 180,E1 -8554.289,E2 -8554.289} C_VEL
LIN {X 0,Y 446.944,Z 575.479,A -85,B 0,C 180,E1 -8555.866,E2 -8555.866} C_VEL
LIN {X 0,Y 447.635,Z 566.603,A -85,B 0,C 180,E1 -8557.215,E2 -8557.215} C_VEL
LIN {X 0,Y 448.376,Z 555.979,A -85,B 0,C 180,E1 -8558.552,E2 -8558.552} C_VEL
LIN {X 0,Y 449.061,Z 545.07,A -85,B 0,C 180,E1 -8559.68,E2 -8559.68} C_VEL
LIN {X 0,Y 449.865,Z 533.101,A -85,B 0,C 180,E1 -8560.691,E2 -8560.691} C_VEL
LIN {X 0,Y 450.511,Z 521.668,A -85,B 0,C 180,E1 -8561.472,E2 -8561.472} C_VEL
LIN {X 0,Y 451.201,Z 508.252,A -85,B 0,C 180,E1 -8562.195,E2 -8562.195} C_VEL
LIN {X 0,Y 451.699,Z 495.057,A -85,B 0,C 180,E1 -8562.724,E2 -8562.724} C_VEL
LIN {X 0,Y 452.034,Z 480.584,A -85,B 0,C 180,E1 -8563.114,E2 -8563.114} C_VEL
LIN {X 0,Y 453.208,Z 365.555,A -85,B 0,C 180,E1 -8564.969,E2 -8564.969} C_VEL
LIN {X 0,Y 449.047,Z 345.554,A -85,B 0,C 180,E1 -8565.517,E2 -8565.517} C_VEL
LIN {X 0,Y 449.011,Z 341.247,A -85,B 0,C 180,E1 -8566.364,E2 -8566.364} C_VEL
LIN {X 0,Y 446.76,Z 329.762,A -85,B 0,C 180,E1 -8568.78,E2 -8568.78} C_VEL
LIN {X 0,Y 446.477,Z 328.499,A -85,B 0,C 180,E1 -8569.067,E2 -8569.067} C_VEL
LIN {X 0,Y 446.421,Z 328.503,A -85,B 0,C 180,E1 -8572.199,E2 -8572.199} C_VEL
LIN {X 0,Y 446.446,Z 328.498,A -85,B 0,C 180,E1 -8575.152,E2 -8575.152} C_VEL
LIN {X 0,Y 446.486,Z 328.491,A -85,B 0,C 180,E1 -8578.178,E2 -8578.178} C_VEL
LIN {X 0,Y 446.42,Z 328.505,A -85,B 0,C 180,E1 -8581.774,E2 -8581.774} C_VEL
LIN {X 0,Y 446.43,Z 328.496,A -85,B 0,C 180,E1 -8584.522,E2 -8584.522} C_VEL
LIN {X 0,Y 446.429,Z 328.499,A -85,B 0,C 180,E1 -8588.081,E2 -8588.081} C_VEL
LIN {X 0,Y 446.424,Z 328.489,A -85,B 0,C 180,E1 -8590.916,E2 -8590.916} C_VEL
LIN {X 0,Y 446.399,Z 328.502,A -85,B 0,C 180,E1 -8593.845,E2 -8593.845} C_VEL
LIN {X 0,Y 446.396,Z 328.502,A -85,B 0,C 180,E1 -8596.402,E2 -8596.402} C_VEL
LIN {X 0,Y 446.422,Z 328.499,A -85,B 0,C 180,E1 -8599.081,E2 -8599.081} C_VEL
LIN {X 0,Y 446.402,Z 328.497,A -85,B 0,C 180,E1 -8602.12,E2 -8602.12} C_VEL
LIN {X 0,Y 446.416,Z 328.501,A -85,B 0,C 180,E1 -8605.475,E2 -8605.475} C_VEL
LIN {X 0,Y 446.407,Z 328.501,A -85,B 0,C 180,E1 -8608.698,E2 -8608.698} C_VEL
LIN {X 0,Y 446.477,Z 328.484,A -85,B 0,C 180,E1 -8611.82,E2 -8611.82} C_VEL
LIN {X 0,Y 446.428,Z 328.499,A -85,B 0,C 180,E1 -8614.845,E2 -8614.845} C_VEL
LIN {X 0,Y 446.438,Z 328.493,A -85,B 0,C 180,E1 -8618.244,E2 -8618.244} C_VEL
LIN {X 0,Y 446.439,Z 328.494,A -85,B 0,C 180,E1 -8621.648,E2 -8621.648} C_VEL
LIN {X 0,Y 446.495,Z 328.492,A -85,B 0,C 180,E1 -8624.479,E2 -8624.479} C_VEL
LIN {X 0,Y 446.503,Z 328.479,A -85,B 0,C 180,E1 -8628.192,E2 -8628.192} C_VEL
LIN {X 0,Y 446.518,Z 328.491,A -85,B 0,C 180,E1 -8630.944,E2 -8630.944} C_VEL
LIN {X 0,Y 446.614,Z 328.47,A -85,B 0,C 180,E1 -8633.676,E2 -8633.676} C_VEL
LIN {X 0,Y 446.65,Z 328.467,A -85,B 0,C 180,E1 -8637.294,E2 -8637.294} C_VEL
LIN {X 0,Y 446.683,Z 328.467,A -85,B 0,C 180,E1 -8640,E2 -8640} C_VEL
LIN {X 0,Y 446.636,Z 328.469,A -85,B 0,C 180,E1 -8642.705,E2 -8642.705} C_VEL
LIN {X 0,Y 446.593,Z 328.483,A -85,B 0,C 180,E1 -8646.324,E2 -8646.324} C_VEL
LIN {X 0,Y 446.507,Z 328.481,A -85,B 0,C 180,E1 -8649.056,E2 -8649.056} C_VEL
LIN {X 0,Y 446.509,Z 328.49,A -85,B 0,C 180,E1 -8652.73,E2 -8652.73} C_VEL
LIN {X 0,Y 446.476,Z 328.494,A -85,B 0,C 180,E1 -8656.459,E2 -8656.459} C_VEL
LIN {X 0,Y 446.456,Z 328.493,A -85,B 0,C 180,E1 -8659.304,E2 -8659.304} C_VEL
LIN {X 0,Y 446.406,Z 328.502,A -85,B 0,C 180,E1 -8662.2,E2 -8662.2} C_VEL
LIN {X 0,Y 446.431,Z 328.494,A -85,B 0,C 180,E1 -8665.154,E2 -8665.154} C_VEL
LIN {X 0,Y 446.438,Z 328.501,A -85,B 0,C 180,E1 -8668.182,E2 -8668.182} C_VEL
LIN {X 0,Y 446.405,Z 328.499,A -85,B 0,C 180,E1 -8671.301,E2 -8671.301} C_VEL
LIN {X 0,Y 446.42,Z 328.499,A -85,B 0,C 180,E1 -8674.524,E2 -8674.524} C_VEL
LIN {X 0,Y 446.407,Z 328.505,A -85,B 0,C 180,E1 -8678.08,E2 -8678.08} C_VEL
LIN {X 0,Y 446.419,Z 328.494,A -85,B 0,C 180,E1 -8680.918,E2 -8680.918} C_VEL
LIN {X 0,Y 446.394,Z 328.507,A -85,B 0,C 180,E1 -8683.847,E2 -8683.847} C_VEL
LIN {X 0,Y 446.393,Z 328.502,A -85,B 0,C 180,E1 -8686.404,E2 -8686.404} C_VEL
LIN {X 0,Y 446.421,Z 328.501,A -85,B 0,C 180,E1 -8689.083,E2 -8689.083} C_VEL
LIN {X 0,Y 446.403,Z 328.506,A -85,B 0,C 180,E1 -8692.122,E2 -8692.122} C_VEL
LIN {X 0,Y 446.427,Z 328.506,A -85,B 0,C 180,E1 -8695.478,E2 -8695.478} C_VEL
LIN {X 0,Y 446.413,Z 328.503,A -85,B 0,C 180,E1 -8698.7,E2 -8698.7} C_VEL
LIN {X 0,Y 446.509,Z 328.644,A -85,B 0,C 180,E1 -8701.488,E2 -8701.488} C_VEL
LIN {X 0,Y 449.744,Z 343.667,A -85,B 0,C 180,E1 -8704.302,E2 -8704.302} C_VEL
LIN {X 0,Y 450.007,Z 347.993,A -85,B 0,C 180,E1 -8705.06,E2 -8705.06} C_VEL
LIN {X 0,Y 448.934,Z 366.558,A -85,B 0,C 180,E1 -8708.174,E2 -8708.174} C_VEL
LIN {X 0,Y 448.776,Z 368.626,A -85,B 0,C 180,E1 -8708.517,E2 -8708.517} C_VEL
LIN {X 0,Y 453.123,Z 393.784,A -85,B 0,C 180,E1 -8709.132,E2 -8709.132} C_VEL
LIN {X 0,Y 451.82,Z 505.942,A -85,B 0,C 180,E1 -8710.935,E2 -8710.935} C_VEL
LIN {X 0,Y 451.359,Z 520.179,A -85,B 0,C 180,E1 -8711.327,E2 -8711.327} C_VEL
LIN {X 0,Y 450.815,Z 534.018,A -85,B 0,C 180,E1 -8711.895,E2 -8711.895} C_VEL
LIN {X 0,Y 450.121,Z 546.984,A -85,B 0,C 180,E1 -8712.605,E2 -8712.605} C_VEL
LIN {X 0,Y 449.312,Z 560.165,A -85,B 0,C 180,E1 -8713.531,E2 -8713.531} C_VEL
LIN {X 0,Y 448.493,Z 571.85,A -85,B 0,C 180,E1 -8714.551,E2 -8714.551} C_VEL
LIN {X 0,Y 447.7,Z 582.554,A -85,B 0,C 180,E1 -8715.686,E2 -8715.686} C_VEL
LIN {X 0,Y 447.072,Z 593.275,A -85,B 0,C 180,E1 -8717.07,E2 -8717.07} C_VEL
LIN {X 0,Y 446.571,Z 601.932,A -85,B 0,C 180,E1 -8718.425,E2 -8718.425} C_VEL
LIN {X 0,Y 446.009,Z 610.321,A -85,B 0,C 180,E1 -8720.019,E2 -8720.019} C_VEL
LIN {X 0,Y 445.767,Z 616.164,A -85,B 0,C 180,E1 -8721.386,E2 -8721.386} C_VEL
LIN {X 0,Y 445.581,Z 620.973,A -85,B 0,C 180,E1 -8722.751,E2 -8722.751} C_VEL
LIN {X 0,Y 445.473,Z 625.946,A -85,B 0,C 180,E1 -8724.568,E2 -8724.568} C_VEL
LIN {X 0,Y 445.37,Z 629.407,A -85,B 0,C 180,E1 -8726.381,E2 -8726.381} C_VEL
LIN {X 0,Y 445.428,Z 630.611,A -85,B 0,C 180,E1 -8727.287,E2 -8727.287} C_VEL
LIN {X 0,Y 445.336,Z 631.99,A -85,B 0,C 180,E1 -8729.096,E2 -8729.096} C_VEL
LIN {X 0,Y 445.336,Z 632.03,A -85,B 0,C 180,E1 -8730.904,E2 -8730.904} C_VEL
LIN {X 0,Y 445.428,Z 630.733,A -85,B 0,C 180,E1 -8732.713,E2 -8732.713} C_VEL
LIN {X 0,Y 445.394,Z 628.062,A -85,B 0,C 180,E1 -8734.525,E2 -8734.525} C_VEL
LIN {X 0,Y 445.528,Z 623.957,A -85,B 0,C 180,E1 -8736.339,E2 -8736.339} C_VEL
LIN {X 0,Y 445.688,Z 618.296,A -85,B 0,C 180,E1 -8738.159,E2 -8738.159} C_VEL
LIN {X 0,Y 446.022,Z 611.925,A -85,B 0,C 180,E1 -8739.752,E2 -8739.752} C_VEL
LIN {X 0,Y 446.515,Z 604.017,A -85,B 0,C 180,E1 -8741.346,E2 -8741.346} C_VEL
LIN {X 0,Y 447.032,Z 595.763,A -85,B 0,C 180,E1 -8742.715,E2 -8742.715} C_VEL
LIN {X 0,Y 447.737,Z 585.837,A -85,B 0,C 180,E1 -8744.081,E2 -8744.081} C_VEL
LIN {X 0,Y 448.518,Z 574.822,A -85,B 0,C 180,E1 -8745.332,E2 -8745.332} C_VEL
LIN {X 0,Y 449.506,Z 562.559,A -85,B 0,C 180,E1 -8746.462,E2 -8746.462} C_VEL
LIN {X 0,Y 450.247,Z 550.926,A -85,B 0,C 180,E1 -8747.335,E2 -8747.335} C_VEL
LIN {X 0,Y 451.031,Z 538.046,A -85,B 0,C 180,E1 -8748.102,E2 -8748.102} C_VEL
LIN {X 0,Y 451.631,Z 524.46,A -85,B 0,C 180,E1 -8748.72,E2 -8748.72} C_VEL
LIN {X 0,Y 452.244,Z 510.387,A -85,B 0,C 180,E1 -8749.164,E2 -8749.164} C_VEL
LIN {X 0,Y 452.59,Z 490.911,A -85,B 0,C 180,E1 -8749.532,E2 -8749.532} C_VEL
LIN {X 0,Y 453.729,Z 393.02,A -85,B 0,C 180,E1 -8751.113,E2 -8751.113} C_VEL
LIN {X 0,Y 449.904,Z 372.305,A -85,B 0,C 180,E1 -8751.668,E2 -8751.668} C_VEL
LIN {X 0,Y 449.155,Z 368.428,A -85,B 0,C 180,E1 -8751.791,E2 -8751.791} C_VEL
LIN {X 0,Y 450.25,Z 351.528,A -85,B 0,C 180,E1 -8754.679,E2 -8754.679} C_VEL
LIN {X 0,Y 450.514,Z 347.005,A -85,B 0,C 180,E1 -8755.462,E2 -8755.462} C_VEL
LIN {X 0,Y 448.296,Z 336.176,A -85,B 0,C 180,E1 -8757.546,E2 -8757.546} C_VEL
LIN {X 0,Y 446.484,Z 328.496,A -85,B 0,C 180,E1 -8759.086,E2 -8759.086} C_VEL
LIN {X 0,Y 446.419,Z 328.505,A -85,B 0,C 180,E1 -8762.361,E2 -8762.361} C_VEL
LIN {X 0,Y 446.417,Z 328.5,A -85,B 0,C 180,E1 -8765.625,E2 -8765.625} C_VEL
LIN {X 0,Y 446.439,Z 328.494,A -85,B 0,C 180,E1 -8769.026,E2 -8769.026} C_VEL
LIN {X 0,Y 446.428,Z 328.5,A -85,B 0,C 180,E1 -8772.276,E2 -8772.276} C_VEL
LIN {X 0,Y 446.447,Z 328.491,A -85,B 0,C 180,E1 -8775.103,E2 -8775.103} C_VEL
LIN {X 0,Y 446.421,Z 328.501,A -85,B 0,C 180,E1 -8778.608,E2 -8778.608} C_VEL
LIN {X 0,Y 446.436,Z 328.498,A -85,B 0,C 180,E1 -8780.972,E2 -8780.972} C_VEL
LIN {X 0,Y 446.411,Z 328.501,A -85,B 0,C 180,E1 -8784.373,E2 -8784.373} C_VEL
LIN {X 0,Y 446.412,Z 328.503,A -85,B 0,C 180,E1 -8787.638,E2 -8787.638} C_VEL
LIN {X 0,Y 446.426,Z 328.488,A -85,B 0,C 180,E1 -8790.789,E2 -8790.789} C_VEL
LIN {X 0,Y 446.428,Z 328.504,A -85,B 0,C 180,E1 -8793.845,E2 -8793.845} C_VEL
LIN {X 0,Y 446.413,Z 328.499,A -85,B 0,C 180,E1 -8796.823,E2 -8796.823} C_VEL
LIN {X 0,Y 446.431,Z 328.498,A -85,B 0,C 180,E1 -8799.737,E2 -8799.737} C_VEL
LIN {X 0,Y 446.442,Z 328.495,A -85,B 0,C 180,E1 -8802.597,E2 -8802.597} C_VEL
LIN {X 0,Y 446.452,Z 328.497,A -85,B 0,C 180,E1 -8805.412,E2 -8805.412} C_VEL
LIN {X 0,Y 446.492,Z 328.486,A -85,B 0,C 180,E1 -8808.193,E2 -8808.193} C_VEL
LIN {X 0,Y 446.492,Z 328.491,A -85,B 0,C 180,E1 -8810.944,E2 -8810.944} C_VEL
LIN {X 0,Y 446.596,Z 328.479,A -85,B 0,C 180,E1 -8813.676,E2 -8813.676} C_VEL
LIN {X 0,Y 446.644,Z 328.472,A -85,B 0,C 180,E1 -8817.295,E2 -8817.295} C_VEL
LIN {X 0,Y 446.684,Z 328.467,A -85,B 0,C 180,E1 -8820,E2 -8820} C_VEL
LIN {X 0,Y 446.667,Z 328.464,A -85,B 0,C 180,E1 -8822.706,E2 -8822.706} C_VEL
LIN {X 0,Y 446.615,Z 328.473,A -85,B 0,C 180,E1 -8826.324,E2 -8826.324} C_VEL
LIN {X 0,Y 446.518,Z 328.489,A -85,B 0,C 180,E1 -8829.056,E2 -8829.056} C_VEL
LIN {X 0,Y 446.511,Z 328.484,A -85,B 0,C 180,E1 -8832.73,E2 -8832.73} C_VEL
LIN {X 0,Y 446.478,Z 328.489,A -85,B 0,C 180,E1 -8836.46,E2 -8836.46} C_VEL
LIN {X 0,Y 446.458,Z 328.496,A -85,B 0,C 180,E1 -8839.304,E2 -8839.304} C_VEL
LIN {X 0,Y 446.408,Z 328.5,A -85,B 0,C 180,E1 -8842.201,E2 -8842.201} C_VEL
LIN {X 0,Y 446.449,Z 328.499,A -85,B 0,C 180,E1 -8845.153,E2 -8845.153} C_VEL
LIN {X 0,Y 446.477,Z 328.49,A -85,B 0,C 180,E1 -8848.18,E2 -8848.18} C_VEL
LIN {X 0,Y 446.412,Z 328.497,A -85,B 0,C 180,E1 -8851.776,E2 -8851.776} C_VEL
LIN {X 0,Y 446.423,Z 328.5,A -85,B 0,C 180,E1 -8854.524,E2 -8854.524} C_VEL
LIN {X 0,Y 446.408,Z 328.499,A -85,B 0,C 180,E1 -8858.08,E2 -8858.08} C_VEL
LIN {X 0,Y 446.422,Z 328.502,A -85,B 0,C 180,E1 -8860.919,E2 -8860.919} C_VEL
LIN {X 0,Y 446.398,Z 328.504,A -85,B 0,C 180,E1 -8863.847,E2 -8863.847} C_VEL
LIN {X 0,Y 446.397,Z 328.507,A -85,B 0,C 180,E1 -8866.404,E2 -8866.404} C_VEL
LIN {X 0,Y 446.425,Z 328.501,A -85,B 0,C 180,E1 -8869.084,E2 -8869.084} C_VEL
LIN {X 0,Y 446.429,Z 328.502,A -85,B 0,C 180,E1 -8871.919,E2 -8871.919} C_VEL
LIN {X 0,Y 446.43,Z 328.496,A -85,B 0,C 180,E1 -8875.478,E2 -8875.478} C_VEL
LIN {X 0,Y 446.449,Z 328.643,A -85,B 0,C 180,E1 -8878.572,E2 -8878.572} C_VEL
LIN {X 0,Y 449.097,Z 340.535,A -85,B 0,C 180,E1 -8881.207,E2 -8881.207} C_VEL
LIN {X 0,Y 449.445,Z 345.306,A -85,B 0,C 180,E1 -8882.192,E2 -8882.192} C_VEL
LIN {X 0,Y 449.414,Z 345.757,A -85,B 0,C 180,E1 -8882.281,E2 -8882.281} C_VEL
LIN {X 0,Y 454.043,Z 366.086,A -85,B 0,C 180,E1 -8882.89,E2 -8882.89} C_VEL
LIN {X 0,Y 452.547,Z 482.124,A -85,B 0,C 180,E1 -8884.78,E2 -8884.78} C_VEL
LIN {X 0,Y 452.119,Z 496.309,A -85,B 0,C 180,E1 -8885.185,E2 -8885.185} C_VEL
LIN {X 0,Y 451.774,Z 505.959,A -85,B 0,C 180,E1 -8885.573,E2 -8885.573} C_VEL
LIN {X 0,Y 450.872,Z 511.526,A -85,B 0,C 180,E1 -8885.801,E2 -8885.801} C_VEL
LIN {X 0,Y 447.695,Z 520.493,A -85,B 0,C 180,E1 -8886.163,E2 -8886.163} C_VEL
LIN {X 0,Y 444.441,Z 529.159,A -85,B 0,C 180,E1 -8886.611,E2 -8886.611} C_VEL
LIN {X 0,Y 443.424,Z 534.248,A -85,B 0,C 180,E1 -8886.971,E2 -8886.971} C_VEL
LIN {X 0,Y 442.586,Z 545.663,A -85,B 0,C 180,E1 -8887.967,E2 -8887.967} C_VEL
LIN {X 0,Y 441.731,Z 555.743,A -85,B 0,C 180,E1 -8889.025,E2 -8889.025} C_VEL
LIN {X 0,Y 441.065,Z 565.1,A -85,B 0,C 180,E1 -8890.202,E2 -8890.202} C_VEL
LIN {X 0,Y 440.289,Z 574.508,A -85,B 0,C 180,E1 -8891.624,E2 -8891.624} C_VEL
LIN {X 0,Y 439.706,Z 582.276,A -85,B 0,C 180,E1 -8893.041,E2 -8893.041} C_VEL
LIN {X 0,Y 439.179,Z 589.643,A -85,B 0,C 180,E1 -8894.69,E2 -8894.69} C_VEL
LIN {X 0,Y 438.823,Z 594.778,A -85,B 0,C 180,E1 -8896.1,E2 -8896.1} C_VEL
LIN {X 0,Y 438.579,Z 599.71,A -85,B 0,C 180,E1 -8897.823,E2 -8897.823} C_VEL
LIN {X 0,Y 438.424,Z 602.111,A -85,B 0,C 180,E1 -8898.91,E2 -8898.91} C_VEL
LIN {X 0,Y 438.254,Z 605.113,A -85,B 0,C 180,E1 -8900.772,E2 -8900.772} C_VEL
LIN {X 0,Y 438.283,Z 606.731,A -85,B 0,C 180,E1 -8902.63,E2 -8902.63} C_VEL
LIN {X 0,Y 438.307,Z 607.015,A -85,B 0,C 180,E1 -8904.479,E2 -8904.479} C_VEL
LIN {X 0,Y 438.288,Z 605.982,A -85,B 0,C 180,E1 -8906.323,E2 -8906.323} C_VEL
LIN {X 0,Y 438.372,Z 604.965,A -85,B 0,C 180,E1 -8907.243,E2 -8907.243} C_VEL
LIN {X 0,Y 438.376,Z 601.923,A -85,B 0,C 180,E1 -8909.081,E2 -8909.081} C_VEL
LIN {X 0,Y 438.49,Z 597.449,A -85,B 0,C 180,E1 -8910.918,E2 -8910.918} C_VEL
LIN {X 0,Y 438.798,Z 591.342,A -85,B 0,C 180,E1 -8912.754,E2 -8912.754} C_VEL
LIN {X 0,Y 439.33,Z 584.53,A -85,B 0,C 180,E1 -8914.358,E2 -8914.358} C_VEL
LIN {X 0,Y 439.921,Z 576.103,A -85,B 0,C 180,E1 -8915.96,E2 -8915.96} C_VEL
LIN {X 0,Y 440.645,Z 567.308,A -85,B 0,C 180,E1 -8917.33,E2 -8917.33} C_VEL
LIN {X 0,Y 441.398,Z 556.823,A -85,B 0,C 180,E1 -8918.683,E2 -8918.683} C_VEL
LIN {X 0,Y 442.141,Z 545.94,A -85,B 0,C 180,E1 -8919.838,E2 -8919.838} C_VEL
LIN {X 0,Y 442.963,Z 534.175,A -85,B 0,C 180,E1 -8920.86,E2 -8920.86} C_VEL
LIN {X 0,Y 443.759,Z 521.192,A -85,B 0,C 180,E1 -8921.765,E2 -8921.765} C_VEL
LIN {X 0,Y 444.408,Z 508.719,A -85,B 0,C 180,E1 -8922.443,E2 -8922.443} C_VEL
LIN {X 0,Y 444.957,Z 494.775,A -85,B 0,C 180,E1 -8923.007,E2 -8923.007} C_VEL
LIN {X 0,Y 445.31,Z 479.964,A -85,B 0,C 180,E1 -8923.403,E2 -8923.403} C_VEL
LIN {X 0,Y 446.527,Z 366.751,A -85,B 0,C 180,E1 -8925.253,E2 -8925.253} C_VEL
LIN {X 0,Y 442.152,Z 345.808,A -85,B 0,C 180,E1 -8925.824,E2 -8925.824} C_VEL
LIN {X 0,Y 441.956,Z 341.811,A -85,B 0,C 180,E1 -8926.632,E2 -8926.632} C_VEL
LIN {X 0,Y 439.715,Z 330.734,A -85,B 0,C 180,E1 -8929.006,E2 -8929.006} C_VEL
LIN {X 0,Y 439.445,Z 329.375,A -85,B 0,C 180,E1 -8929.336,E2 -8929.336} C_VEL
LIN {X 0,Y 439.367,Z 329.379,A -85,B 0,C 180,E1 -8932.575,E2 -8932.575} C_VEL
LIN {X 0,Y 439.4,Z 329.379,A -85,B 0,C 180,E1 -8935.584,E2 -8935.584} C_VEL
LIN {X 0,Y 439.419,Z 329.369,A -85,B 0,C 180,E1 -8938.672,E2 -8938.672} C_VEL
LIN {X 0,Y 439.371,Z 329.38,A -85,B 0,C 180,E1 -8942.029,E2 -8942.029} C_VEL
LIN {X 0,Y 439.396,Z 329.374,A -85,B 0,C 180,E1 -8945.34,E2 -8945.34} C_VEL
LIN {X 0,Y 439.387,Z 329.374,A -85,B 0,C 180,E1 -8948.593,E2 -8948.593} C_VEL
LIN {X 0,Y 439.386,Z 329.369,A -85,B 0,C 180,E1 -8951.256,E2 -8951.256} C_VEL
LIN {X 0,Y 439.398,Z 329.372,A -85,B 0,C 180,E1 -8954.728,E2 -8954.728} C_VEL
LIN {X 0,Y 439.391,Z 329.373,A -85,B 0,C 180,E1 -8957.794,E2 -8957.794} C_VEL
LIN {X 0,Y 439.39,Z 329.374,A -85,B 0,C 180,E1 -8960.223,E2 -8960.223} C_VEL
LIN {X 0,Y 439.367,Z 329.38,A -85,B 0,C 180,E1 -8963.712,E2 -8963.712} C_VEL
LIN {X 0,Y 439.365,Z 329.378,A -85,B 0,C 180,E1 -8967.053,E2 -8967.053} C_VEL
LIN {X 0,Y 439.373,Z 329.376,A -85,B 0,C 180,E1 -8970.273,E2 -8970.273} C_VEL
LIN {X 0,Y 439.41,Z 329.372,A -85,B 0,C 180,E1 -8973.395,E2 -8973.395} C_VEL
LIN {X 0,Y 439.372,Z 329.378,A -85,B 0,C 180,E1 -8976.428,E2 -8976.428} C_VEL
LIN {X 0,Y 439.377,Z 329.367,A -85,B 0,C 180,E1 -8979.396,E2 -8979.396} C_VEL
LIN {X 0,Y 439.393,Z 329.373,A -85,B 0,C 180,E1 -8982.308,E2 -8982.308} C_VEL
LIN {X 0,Y 439.433,Z 329.367,A -85,B 0,C 180,E1 -8985.173,E2 -8985.173} C_VEL
LIN {X 0,Y 439.47,Z 329.353,A -85,B 0,C 180,E1 -8988.001,E2 -8988.001} C_VEL
LIN {X 0,Y 439.491,Z 329.361,A -85,B 0,C 180,E1 -8991.725,E2 -8991.725} C_VEL
LIN {X 0,Y 439.594,Z 329.345,A -85,B 0,C 180,E1 -8994.495,E2 -8994.495} C_VEL
LIN {X 0,Y 439.617,Z 329.345,A -85,B 0,C 180,E1 -8998.167,E2 -8998.167} C_VEL
LIN {X 0,Y 439.571,Z 329.352,A -85,B 0,C 180,E1 -9000.916,E2 -9000.916} C_VEL
LIN {X 0,Y 439.587,Z 329.346,A -85,B 0,C 180,E1 -9002.749,E2 -9002.749} C_VEL
LIN {X 0,Y 439.546,Z 329.362,A -85,B 0,C 180,E1 -9006.426,E2 -9006.426} C_VEL
LIN {X 0,Y 439.472,Z 329.356,A -85,B 0,C 180,E1 -9009.202,E2 -9009.202} C_VEL
LIN {X 0,Y 439.453,Z 329.367,A -85,B 0,C 180,E1 -9012.938,E2 -9012.938} C_VEL
LIN {X 0,Y 439.434,Z 329.369,A -85,B 0,C 180,E1 -9016.348,E2 -9016.348} C_VEL
LIN {X 0,Y 439.39,Z 329.375,A -85,B 0,C 180,E1 -9019.627,E2 -9019.627} C_VEL
LIN {X 0,Y 439.352,Z 329.38,A -85,B 0,C 180,E1 -9022.576,E2 -9022.576} C_VEL
LIN {X 0,Y 439.368,Z 329.376,A -85,B 0,C 180,E1 -9025.587,E2 -9025.587} C_VEL
LIN {X 0,Y 439.389,Z 329.374,A -85,B 0,C 180,E1 -9028.675,E2 -9028.675} C_VEL
LIN {X 0,Y 439.36,Z 329.384,A -85,B 0,C 180,E1 -9032.031,E2 -9032.031} C_VEL
LIN {X 0,Y 439.386,Z 329.375,A -85,B 0,C 180,E1 -9035.341,E2 -9035.341} C_VEL
LIN {X 0,Y 439.377,Z 329.377,A -85,B 0,C 180,E1 -9038.595,E2 -9038.595} C_VEL
LIN {X 0,Y 439.381,Z 329.373,A -85,B 0,C 180,E1 -9041.257,E2 -9041.257} C_VEL
LIN {X 0,Y 439.394,Z 329.373,A -85,B 0,C 180,E1 -9044.73,E2 -9044.73} C_VEL
LIN {X 0,Y 439.39,Z 329.38,A -85,B 0,C 180,E1 -9047.796,E2 -9047.796} C_VEL
LIN {X 0,Y 439.389,Z 329.379,A -85,B 0,C 180,E1 -9050.225,E2 -9050.225} C_VEL
LIN {X 0,Y 439.37,Z 329.385,A -85,B 0,C 180,E1 -9053.714,E2 -9053.714} C_VEL
LIN {X 0,Y 439.369,Z 329.383,A -85,B 0,C 180,E1 -9057.055,E2 -9057.055} C_VEL
LIN {X 0,Y 439.421,Z 329.375,A -85,B 0,C 180,E1 -9060.804,E2 -9060.804} C_VEL
LIN {X 0,Y 439.443,Z 329.415,A -85,B 0,C 180,E1 -9061.199,E2 -9061.199} C_VEL
LIN {X 0,Y 442.443,Z 343.268,A -85,B 0,C 180,E1 -9063.846,E2 -9063.846} C_VEL
LIN {X 0,Y 443.173,Z 347.791,A -85,B 0,C 180,E1 -9064.679,E2 -9064.679} C_VEL
LIN {X 0,Y 442.06,Z 366.185,A -85,B 0,C 180,E1 -9067.817,E2 -9067.817} C_VEL
LIN {X 0,Y 441.934,Z 368.589,A -85,B 0,C 180,E1 -9068.205,E2 -9068.205} C_VEL
LIN {X 0,Y 446.42,Z 394.773,A -85,B 0,C 180,E1 -9068.851,E2 -9068.851} C_VEL
LIN {X 0,Y 445.062,Z 505.904,A -85,B 0,C 180,E1 -9070.664,E2 -9070.664} C_VEL
LIN {X 0,Y 444.592,Z 520.072,A -85,B 0,C 180,E1 -9071.062,E2 -9071.062} C_VEL
LIN {X 0,Y 444.011,Z 533.572,A -85,B 0,C 180,E1 -9071.621,E2 -9071.621} C_VEL
LIN {X 0,Y 443.28,Z 546.703,A -85,B 0,C 180,E1 -9072.349,E2 -9072.349} C_VEL
LIN {X 0,Y 442.423,Z 559.653,A -85,B 0,C 180,E1 -9073.267,E2 -9073.267} C_VEL
LIN {X 0,Y 441.603,Z 571.399,A -85,B 0,C 180,E1 -9074.303,E2 -9074.303} C_VEL
LIN {X 0,Y 440.76,Z 582.147,A -85,B 0,C 180,E1 -9075.456,E2 -9075.456} C_VEL
LIN {X 0,Y 440.09,Z 592.97,A -85,B 0,C 180,E1 -9076.87,E2 -9076.87} C_VEL
LIN {X 0,Y 439.552,Z 601.593,A -85,B 0,C 180,E1 -9078.238,E2 -9078.238} C_VEL
LIN {X 0,Y 438.963,Z 610.012,A -85,B 0,C 180,E1 -9079.857,E2 -9079.857} C_VEL
LIN {X 0,Y 438.69,Z 615.874,A -85,B 0,C 180,E1 -9081.246,E2 -9081.246} C_VEL
LIN {X 0,Y 438.491,Z 622.136,A -85,B 0,C 180,E1 -9083.096,E2 -9083.096} C_VEL
LIN {X 0,Y 438.373,Z 625.694,A -85,B 0,C 180,E1 -9084.48,E2 -9084.48} C_VEL
LIN {X 0,Y 438.271,Z 629.172,A -85,B 0,C 180,E1 -9086.322,E2 -9086.322} C_VEL
LIN {X 0,Y 438.336,Z 630.384,A -85,B 0,C 180,E1 -9087.243,E2 -9087.243} C_VEL
LIN {X 0,Y 438.25,Z 631.778,A -85,B 0,C 180,E1 -9089.081,E2 -9089.081} C_VEL
LIN {X 0,Y 438.25,Z 631.834,A -85,B 0,C 180,E1 -9090.919,E2 -9090.919} C_VEL
LIN {X 0,Y 438.336,Z 630.554,A -85,B 0,C 180,E1 -9092.757,E2 -9092.757} C_VEL
LIN {X 0,Y 438.319,Z 627.902,A -85,B 0,C 180,E1 -9094.598,E2 -9094.598} C_VEL
LIN {X 0,Y 438.446,Z 623.813,A -85,B 0,C 180,E1 -9096.442,E2 -9096.442} C_VEL
LIN {X 0,Y 438.623,Z 618.171,A -85,B 0,C 180,E1 -9098.291,E2 -9098.291} C_VEL
LIN {X 0,Y 438.982,Z 611.822,A -85,B 0,C 180,E1 -9099.91,E2 -9099.91} C_VEL
LIN {X 0,Y 439.518,Z 603.938,A -85,B 0,C 180,E1 -9101.53,E2 -9101.53} C_VEL
LIN {X 0,Y 440.128,Z 594.677,A -85,B 0,C 180,E1 -9103.081,E2 -9103.081} C_VEL
LIN {X 0,Y 440.8,Z 585.822,A -85,B 0,C 180,E1 -9104.307,E2 -9104.307} C_VEL
LIN {X 0,Y 441.656,Z 574.849,A -85,B 0,C 180,E1 -9105.576,E2 -9105.576} C_VEL
LIN {X 0,Y 442.702,Z 562.663,A -85,B 0,C 180,E1 -9106.722,E2 -9106.722} C_VEL
LIN {X 0,Y 443.562,Z 550.051,A -85,B 0,C 180,E1 -9107.677,E2 -9107.677} C_VEL
LIN {X 0,Y 444.36,Z 537.279,A -85,B 0,C 180,E1 -9108.44,E2 -9108.44} C_VEL
LIN {X 0,Y 444.96,Z 524.185,A -85,B 0,C 180,E1 -9109.041,E2 -9109.041} C_VEL
LIN {X 0,Y 445.604,Z 510.082,A -85,B 0,C 180,E1 -9109.491,E2 -9109.491} C_VEL
LIN {X 0,Y 445.991,Z 490.552,A -85,B 0,C 180,E1 -9109.863,E2 -9109.863} C_VEL
LIN {X 0,Y 447.215,Z 394.453,A -85,B 0,C 180,E1 -9111.436,E2 -9111.436} C_VEL
LIN {X 0,Y 443.364,Z 373.311,A -85,B 0,C 180,E1 -9112.013,E2 -9112.013} C_VEL
LIN {X 0,Y 442.328,Z 368.15,A -85,B 0,C 180,E1 -9112.188,E2 -9112.188} C_VEL
LIN {X 0,Y 443.511,Z 351.52,A -85,B 0,C 180,E1 -9115.08,E2 -9115.08} C_VEL
LIN {X 0,Y 443.677,Z 348.731,A -85,B 0,C 180,E1 -9115.571,E2 -9115.571} C_VEL
LIN {X 0,Y 441.368,Z 337.583,A -85,B 0,C 180,E1 -9117.758,E2 -9117.758} C_VEL
LIN {X 0,Y 439.415,Z 329.376,A -85,B 0,C 180,E1 -9119.459,E2 -9119.459} C_VEL
LIN {X 0,Y 439.369,Z 329.382,A -85,B 0,C 180,E1 -9122.945,E2 -9122.945} C_VEL
LIN {X 0,Y 439.37,Z 329.38,A -85,B 0,C 180,E1 -9126.286,E2 -9126.286} C_VEL
LIN {X 0,Y 439.396,Z 329.371,A -85,B 0,C 180,E1 -9129.848,E2 -9129.848} C_VEL
LIN {X 0,Y 439.375,Z 329.375,A -85,B 0,C 180,E1 -9132.626,E2 -9132.626} C_VEL
LIN {X 0,Y 439.394,Z 329.369,A -85,B 0,C 180,E1 -9135.27,E2 -9135.27} C_VEL
LIN {X 0,Y 439.381,Z 329.377,A -85,B 0,C 180,E1 -9138.743,E2 -9138.743} C_VEL
LIN {X 0,Y 439.366,Z 329.38,A -85,B 0,C 180,E1 -9141.607,E2 -9141.607} C_VEL
LIN {X 0,Y 439.391,Z 329.372,A -85,B 0,C 180,E1 -9144.843,E2 -9144.843} C_VEL
LIN {X 0,Y 439.363,Z 329.375,A -85,B 0,C 180,E1 -9148.139,E2 -9148.139} C_VEL
LIN {X 0,Y 439.398,Z 329.366,A -85,B 0,C 180,E1 -9151.604,E2 -9151.604} C_VEL
LIN {X 0,Y 439.367,Z 329.376,A -85,B 0,C 180,E1 -9154.413,E2 -9154.413} C_VEL
LIN {X 0,Y 439.352,Z 329.381,A -85,B 0,C 180,E1 -9157.424,E2 -9157.424} C_VEL
LIN {X 0,Y 439.429,Z 329.369,A -85,B 0,C 180,E1 -9160.663,E2 -9160.663} C_VEL
LIN {X 0,Y 439.449,Z 329.367,A -85,B 0,C 180,E1 -9164.224,E2 -9164.224} C_VEL
LIN {X 0,Y 439.462,Z 329.363,A -85,B 0,C 180,E1 -9168.001,E2 -9168.001} C_VEL
LIN {X 0,Y 439.466,Z 329.366,A -85,B 0,C 180,E1 -9171.725,E2 -9171.725} C_VEL
LIN {X 0,Y 439.588,Z 329.349,A -85,B 0,C 180,E1 -9174.496,E2 -9174.496} C_VEL
LIN {X 0,Y 439.612,Z 329.343,A -85,B 0,C 180,E1 -9178.168,E2 -9178.168} C_VEL
LIN {X 0,Y 439.636,Z 329.345,A -85,B 0,C 180,E1 -9180,E2 -9180} C_VEL
LIN {X 0,Y 439.616,Z 329.343,A -85,B 0,C 180,E1 -9182.749,E2 -9182.749} C_VEL
LIN {X 0,Y 439.586,Z 329.349,A -85,B 0,C 180,E1 -9186.426,E2 -9186.426} C_VEL
LIN {X 0,Y 439.482,Z 329.368,A -85,B 0,C 180,E1 -9189.202,E2 -9189.202} C_VEL
LIN {X 0,Y 439.454,Z 329.365,A -85,B 0,C 180,E1 -9192.938,E2 -9192.938} C_VEL
LIN {X 0,Y 439.436,Z 329.366,A -85,B 0,C 180,E1 -9196.349,E2 -9196.349} C_VEL
LIN {X 0,Y 439.392,Z 329.373,A -85,B 0,C 180,E1 -9199.627,E2 -9199.627} C_VEL
LIN {X 0,Y 439.355,Z 329.382,A -85,B 0,C 180,E1 -9202.576,E2 -9202.576} C_VEL
LIN {X 0,Y 439.397,Z 329.374,A -85,B 0,C 180,E1 -9205.586,E2 -9205.586} C_VEL
LIN {X 0,Y 439.41,Z 329.374,A -85,B 0,C 180,E1 -9208.675,E2 -9208.675} C_VEL
LIN {X 0,Y 439.363,Z 329.376,A -85,B 0,C 180,E1 -9212.031,E2 -9212.031} C_VEL
LIN {X 0,Y 439.388,Z 329.375,A -85,B 0,C 180,E1 -9215.341,E2 -9215.341} C_VEL
LIN {X 0,Y 439.37,Z 329.382,A -85,B 0,C 180,E1 -9218.597,E2 -9218.597} C_VEL
LIN {X 0,Y 439.384,Z 329.376,A -85,B 0,C 180,E1 -9221.258,E2 -9221.258} C_VEL
LIN {X 0,Y 439.398,Z 329.377,A -85,B 0,C 180,E1 -9224.73,E2 -9224.73} C_VEL
LIN {X 0,Y 439.394,Z 329.377,A -85,B 0,C 180,E1 -9227.797,E2 -9227.797} C_VEL
LIN {X 0,Y 439.435,Z 329.374,A -85,B 0,C 180,E1 -9230.23,E2 -9230.23} C_VEL
LIN {X 0,Y 439.376,Z 329.379,A -85,B 0,C 180,E1 -9233.714,E2 -9233.714} C_VEL
LIN {X 0,Y 439.373,Z 329.382,A -85,B 0,C 180,E1 -9237.055,E2 -9237.055} C_VEL
LIN {X 0,Y 439.399,Z 329.528,A -85,B 0,C 180,E1 -9238.244,E2 -9238.244} C_VEL
LIN {X 0,Y 441.942,Z 340.776,A -85,B 0,C 180,E1 -9240.788,E2 -9240.788} C_VEL
LIN {X 0,Y 442.594,Z 345.969,A -85,B 0,C 180,E1 -9241.897,E2 -9241.897} C_VEL
LIN {X 0,Y 447.066,Z 365.06,A -85,B 0,C 180,E1 -9242.492,E2 -9242.492} C_VEL
LIN {X 0,Y 447.529,Z 367.424,A -85,B 0,C 180,E1 -9242.558,E2 -9242.558} C_VEL
LIN {X 0,Y 445.926,Z 482.624,A -85,B 0,C 180,E1 -9244.463,E2 -9244.463} C_VEL
LIN {X 0,Y 445.457,Z 496.946,A -85,B 0,C 180,E1 -9244.882,E2 -9244.882} C_VEL
LIN {X 0,Y 444.89,Z 511.21,A -85,B 0,C 180,E1 -9245.502,E2 -9245.502} C_VEL
LIN {X 0,Y 444.149,Z 523.476,A -85,B 0,C 180,E1 -9246.204,E2 -9246.204} C_VEL
LIN {X 0,Y 443.424,Z 534.248,A -85,B 0,C 180,E1 -9246.971,E2 -9246.971} C_VEL
LIN {X 0,Y 442.403,Z 539.32,A -85,B 0,C 180,E1 -9247.357,E2 -9247.357} C_VEL
LIN {X 0,Y 439.035,Z 547.322,A -85,B 0,C 180,E1 -9247.979,E2 -9247.979} C_VEL
LIN {X 0,Y 435.701,Z 554.968,A -85,B 0,C 180,E1 -9248.672,E2 -9248.672} C_VEL
LIN {X 0,Y 434.713,Z 559.336,A -85,B 0,C 180,E1 -9249.17,E2 -9249.17} C_VEL
LIN {X 0,Y 433.788,Z 569.782,A -85,B 0,C 180,E1 -9250.602,E2 -9250.602} C_VEL
LIN {X 0,Y 433.045,Z 578.385,A -85,B 0,C 180,E1 -9252.04,E2 -9252.04} C_VEL
LIN {X 0,Y 432.441,Z 586.243,A -85,B 0,C 180,E1 -9253.645,E2 -9253.645} C_VEL
LIN {X 0,Y 431.89,Z 593.107,A -85,B 0,C 180,E1 -9255.391,E2 -9255.391} C_VEL
LIN {X 0,Y 431.566,Z 598.887,A -85,B 0,C 180,E1 -9257.301,E2 -9257.301} C_VEL
LIN {X 0,Y 431.365,Z 602.173,A -85,B 0,C 180,E1 -9258.726,E2 -9258.726} C_VEL
LIN {X 0,Y 431.163,Z 605.228,A -85,B 0,C 180,E1 -9260.619,E2 -9260.619} C_VEL
LIN {X 0,Y 431.185,Z 606.896,A -85,B 0,C 180,E1 -9262.508,E2 -9262.508} C_VEL
LIN {X 0,Y 431.216,Z 607.23,A -85,B 0,C 180,E1 -9264.388,E2 -9264.388} C_VEL
LIN {X 0,Y 431.191,Z 606.246,A -85,B 0,C 180,E1 -9266.262,E2 -9266.262} C_VEL
LIN {X 0,Y 431.257,Z 603.932,A -85,B 0,C 180,E1 -9268.132,E2 -9268.132} C_VEL
LIN {X 0,Y 431.361,Z 600.238,A -85,B 0,C 180,E1 -9270,E2 -9270} C_VEL
LIN {X 0,Y 431.552,Z 595.054,A -85,B 0,C 180,E1 -9271.866,E2 -9271.866} C_VEL
LIN {X 0,Y 431.896,Z 590.028,A -85,B 0,C 180,E1 -9273.265,E2 -9273.265} C_VEL
LIN {X 0,Y 432.407,Z 582.87,A -85,B 0,C 180,E1 -9274.895,E2 -9274.895} C_VEL
LIN {X 0,Y 433.049,Z 575.375,A -85,B 0,C 180,E1 -9276.289,E2 -9276.289} C_VEL
LIN {X 0,Y 433.771,Z 566.397,A -85,B 0,C 180,E1 -9277.681,E2 -9277.681} C_VEL
LIN {X 0,Y 434.612,Z 555.631,A -85,B 0,C 180,E1 -9279.061,E2 -9279.061} C_VEL
LIN {X 0,Y 435.396,Z 544.511,A -85,B 0,C 180,E1 -9280.227,E2 -9280.227} C_VEL
LIN {X 0,Y 436.242,Z 532.332,A -85,B 0,C 180,E1 -9281.264,E2 -9281.264} C_VEL
LIN {X 0,Y 436.968,Z 520.656,A -85,B 0,C 180,E1 -9282.068,E2 -9282.068} C_VEL
LIN {X 0,Y 437.672,Z 507.952,A -85,B 0,C 180,E1 -9282.755,E2 -9282.755} C_VEL
LIN {X 0,Y 438.234,Z 494.434,A -85,B 0,C 180,E1 -9283.299,E2 -9283.299} C_VEL
LIN {X 0,Y 438.552,Z 480.769,A -85,B 0,C 180,E1 -9283.672,E2 -9283.672} C_VEL
LIN {X 0,Y 439.911,Z 368.422,A -85,B 0,C 180,E1 -9285.533,E2 -9285.533} C_VEL
LIN {X 0,Y 435.265,Z 346.074,A -85,B 0,C 180,E1 -9286.142,E2 -9286.142} C_VEL
LIN {X 0,Y 434.452,Z 340.284,A -85,B 0,C 180,E1 -9287.363,E2 -9287.363} C_VEL
LIN {X 0,Y 432.391,Z 330.255,A -85,B 0,C 180,E1 -9289.585,E2 -9289.585} C_VEL
LIN {X 0,Y 432.321,Z 330.257,A -85,B 0,C 180,E1 -9292.963,E2 -9292.963} C_VEL
LIN {X 0,Y 432.363,Z 330.256,A -85,B 0,C 180,E1 -9296.032,E2 -9296.032} C_VEL
LIN {X 0,Y 432.344,Z 330.251,A -85,B 0,C 180,E1 -9299.186,E2 -9299.186} C_VEL
LIN {X 0,Y 432.323,Z 330.255,A -85,B 0,C 180,E1 -9302.442,E2 -9302.442} C_VEL
LIN {X 0,Y 432.345,Z 330.251,A -85,B 0,C 180,E1 -9305.631,E2 -9305.631} C_VEL
LIN {X 0,Y 432.349,Z 330.251,A -85,B 0,C 180,E1 -9308.715,E2 -9308.715} C_VEL
LIN {X 0,Y 432.332,Z 330.257,A -85,B 0,C 180,E1 -9311.796,E2 -9311.796} C_VEL
LIN {X 0,Y 432.331,Z 330.252,A -85,B 0,C 180,E1 -9314.346,E2 -9314.346} C_VEL
LIN {X 0,Y 432.316,Z 330.259,A -85,B 0,C 180,E1 -9317.014,E2 -9317.014} C_VEL
LIN {X 0,Y 432.328,Z 330.256,A -85,B 0,C 180,E1 -9319.82,E2 -9319.82} C_VEL
LIN {X 0,Y 432.3,Z 330.257,A -85,B 0,C 180,E1 -9323.021,E2 -9323.021} C_VEL
LIN {X 0,Y 432.351,Z 330.248,A -85,B 0,C 180,E1 -9325.996,E2 -9325.996} C_VEL
LIN {X 0,Y 432.339,Z 330.255,A -85,B 0,C 180,E1 -9329.489,E2 -9329.489} C_VEL
LIN {X 0,Y 432.377,Z 330.243,A -85,B 0,C 180,E1 -9332.927,E2 -9332.927} C_VEL
LIN {X 0,Y 432.356,Z 330.25,A -85,B 0,C 180,E1 -9336.022,E2 -9336.022} C_VEL
LIN {X 0,Y 432.339,Z 330.246,A -85,B 0,C 180,E1 -9339.045,E2 -9339.045} C_VEL
LIN {X 0,Y 432.349,Z 330.249,A -85,B 0,C 180,E1 -9342.009,E2 -9342.009} C_VEL
LIN {X 0,Y 432.382,Z 330.248,A -85,B 0,C 180,E1 -9344.926,E2 -9344.926} C_VEL
LIN {X 0,Y 432.447,Z 330.228,A -85,B 0,C 180,E1 -9347.803,E2 -9347.803} C_VEL
LIN {X 0,Y 432.451,Z 330.238,A -85,B 0,C 180,E1 -9351.589,E2 -9351.589} C_VEL
LIN {X 0,Y 432.571,Z 330.22,A -85,B 0,C 180,E1 -9354.405,E2 -9354.405} C_VEL
LIN {X 0,Y 432.586,Z 330.22,A -85,B 0,C 180,E1 -9358.138,E2 -9358.138} C_VEL
LIN {X 0,Y 432.532,Z 330.228,A -85,B 0,C 180,E1 -9360.931,E2 -9360.931} C_VEL
LIN {X 0,Y 432.541,Z 330.223,A -85,B 0,C 180,E1 -9362.794,E2 -9362.794} C_VEL
LIN {X 0,Y 432.539,Z 330.227,A -85,B 0,C 180,E1 -9365.594,E2 -9365.594} C_VEL
LIN {X 0,Y 432.437,Z 330.24,A -85,B 0,C 180,E1 -9368.41,E2 -9368.41} C_VEL
LIN {X 0,Y 432.446,Z 330.244,A -85,B 0,C 180,E1 -9372.197,E2 -9372.197} C_VEL
LIN {X 0,Y 432.418,Z 330.24,A -85,B 0,C 180,E1 -9376.039,E2 -9376.039} C_VEL
LIN {X 0,Y 432.375,Z 330.248,A -85,B 0,C 180,E1 -9379.485,E2 -9379.485} C_VEL
LIN {X 0,Y 432.306,Z 330.255,A -85,B 0,C 180,E1 -9382.965,E2 -9382.965} C_VEL
LIN {X 0,Y 432.328,Z 330.251,A -85,B 0,C 180,E1 -9385.002,E2 -9385.002} C_VEL
LIN {X 0,Y 432.337,Z 330.258,A -85,B 0,C 180,E1 -9388.126,E2 -9388.126} C_VEL
LIN {X 0,Y 432.311,Z 330.255,A -85,B 0,C 180,E1 -9391.347,E2 -9391.347} C_VEL
LIN {X 0,Y 432.331,Z 330.253,A -85,B 0,C 180,E1 -9394.678,E2 -9394.678} C_VEL
LIN {X 0,Y 432.331,Z 330.258,A -85,B 0,C 180,E1 -9398.15,E2 -9398.15} C_VEL
LIN {X 0,Y 432.325,Z 330.251,A -85,B 0,C 180,E1 -9401.603,E2 -9401.603} C_VEL
LIN {X 0,Y 432.327,Z 330.255,A -85,B 0,C 180,E1 -9404.348,E2 -9404.348} C_VEL
LIN {X 0,Y 432.314,Z 330.257,A -85,B 0,C 180,E1 -9407.016,E2 -9407.016} C_VEL
LIN {X 0,Y 432.328,Z 330.26,A -85,B 0,C 180,E1 -9409.822,E2 -9409.822} C_VEL
LIN {X 0,Y 432.302,Z 330.263,A -85,B 0,C 180,E1 -9413.023,E2 -9413.023} C_VEL
LIN {X 0,Y 432.356,Z 330.256,A -85,B 0,C 180,E1 -9415.997,E2 -9415.997} C_VEL
LIN {X 0,Y 432.344,Z 330.257,A -85,B 0,C 180,E1 -9419.49,E2 -9419.49} C_VEL
LIN {X 0,Y 432.42,Z 330.337,A -85,B 0,C 180,E1 -9420.93,E2 -9420.93} C_VEL
LIN {X 0,Y 435.438,Z 344.311,A -85,B 0,C 180,E1 -9423.651,E2 -9423.651} C_VEL
LIN {X 0,Y 436.27,Z 349.386,A -85,B 0,C 180,E1 -9424.602,E2 -9424.602} C_VEL
LIN {X 0,Y 435.039,Z 368.138,A -85,B 0,C 180,E1 -9427.85,E2 -9427.85} C_VEL
LIN {X 0,Y 439.737,Z 395.389,A -85,B 0,C 180,E1 -9428.557,E2 -9428.557} C_VEL
LIN {X 0,Y 438.317,Z 505.796,A -85,B 0,C 180,E1 -9430.385,E2 -9430.385} C_VEL
LIN {X 0,Y 437.829,Z 519.927,A -85,B 0,C 180,E1 -9430.789,E2 -9430.789} C_VEL
LIN {X 0,Y 437.217,Z 532.908,A -85,B 0,C 180,E1 -9431.329,E2 -9431.329} C_VEL
LIN {X 0,Y 436.456,Z 546.399,A -85,B 0,C 180,E1 -9432.084,E2 -9432.084} C_VEL
LIN {X 0,Y 435.597,Z 559.125,A -85,B 0,C 180,E1 -9432.997,E2 -9432.997} C_VEL
LIN {X 0,Y 434.693,Z 570.929,A -85,B 0,C 180,E1 -9434.047,E2 -9434.047} C_VEL
LIN {X 0,Y 433.83,Z 581.726,A -85,B 0,C 180,E1 -9435.218,E2 -9435.218} C_VEL
LIN {X 0,Y 433.136,Z 592.423,A -85,B 0,C 180,E1 -9436.632,E2 -9436.632} C_VEL
LIN {X 0,Y 432.514,Z 601.242,A -85,B 0,C 180,E1 -9438.043,E2 -9438.043} C_VEL
LIN {X 0,Y 431.929,Z 609.693,A -85,B 0,C 180,E1 -9439.69,E2 -9439.69} C_VEL
LIN {X 0,Y 431.616,Z 615.576,A -85,B 0,C 180,E1 -9441.102,E2 -9441.102} C_VEL
LIN {X 0,Y 431.406,Z 621.864,A -85,B 0,C 180,E1 -9442.982,E2 -9442.982} C_VEL
LIN {X 0,Y 431.277,Z 625.438,A -85,B 0,C 180,E1 -9444.389,E2 -9444.389} C_VEL
LIN {X 0,Y 431.177,Z 628.934,A -85,B 0,C 180,E1 -9446.262,E2 -9446.262} C_VEL
LIN {X 0,Y 431.2,Z 631.028,A -85,B 0,C 180,E1 -9448.132,E2 -9448.132} C_VEL
LIN {X 0,Y 431.165,Z 631.768,A -85,B 0,C 180,E1 -9450,E2 -9450} C_VEL
LIN {X 0,Y 431.2,Z 631.175,A -85,B 0,C 180,E1 -9451.868,E2 -9451.868} C_VEL
LIN {X 0,Y 431.176,Z 629.234,A -85,B 0,C 180,E1 -9453.738,E2 -9453.738} C_VEL
LIN {X 0,Y 431.278,Z 625.895,A -85,B 0,C 180,E1 -9455.611,E2 -9455.611} C_VEL
LIN {X 0,Y 431.391,Z 622.423,A -85,B 0,C 180,E1 -9457.018,E2 -9457.018} C_VEL
LIN {X 0,Y 431.661,Z 616.423,A -85,B 0,C 180,E1 -9458.898,E2 -9458.898} C_VEL
LIN {X 0,Y 432.059,Z 609.683,A -85,B 0,C 180,E1 -9460.544,E2 -9460.544} C_VEL
LIN {X 0,Y 432.733,Z 601.313,A -85,B 0,C 180,E1 -9462.188,E2 -9462.188} C_VEL
LIN {X 0,Y 433.322,Z 592.933,A -85,B 0,C 180,E1 -9463.554,E2 -9463.554} C_VEL
LIN {X 0,Y 434.209,Z 582.078,A -85,B 0,C 180,E1 -9465.009,E2 -9465.009} C_VEL
LIN {X 0,Y 435.112,Z 571.483,A -85,B 0,C 180,E1 -9466.178,E2 -9466.178} C_VEL
LIN {X 0,Y 436.073,Z 559.95,A -85,B 0,C 180,E1 -9467.226,E2 -9467.226} C_VEL
LIN {X 0,Y 437.067,Z 546.448,A -85,B 0,C 180,E1 -9468.211,E2 -9468.211} C_VEL
LIN {X 0,Y 437.883,Z 533.108,A -85,B 0,C 180,E1 -9468.966,E2 -9468.966} C_VEL
LIN {X 0,Y 438.586,Z 520.148,A -85,B 0,C 180,E1 -9469.511,E2 -9469.511} C_VEL
LIN {X 0,Y 439.13,Z 506.426,A -85,B 0,C 180,E1 -9469.912,E2 -9469.912} C_VEL
LIN {X 0,Y 440.656,Z 395.285,A -85,B 0,C 180,E1 -9471.784,E2 -9471.784} C_VEL
LIN {X 0,Y 437.073,Z 375.493,A -85,B 0,C 180,E1 -9472.335,E2 -9472.335} C_VEL
LIN {X 0,Y 435.522,Z 368.03,A -85,B 0,C 180,E1 -9472.573,E2 -9472.573} C_VEL
LIN {X 0,Y 436.795,Z 351.243,A -85,B 0,C 180,E1 -9475.543,E2 -9475.543} C_VEL
LIN {X 0,Y 435.992,Z 345.947,A -85,B 0,C 180,E1 -9476.571,E2 -9476.571} C_VEL
LIN {X 0,Y 433.154,Z 333.443,A -85,B 0,C 180,E1 -9479.127,E2 -9479.127} C_VEL
LIN {X 0,Y 432.371,Z 330.254,A -85,B 0,C 180,E1 -9479.82,E2 -9479.82} C_VEL
LIN {X 0,Y 432.336,Z 330.257,A -85,B 0,C 180,E1 -9483.551,E2 -9483.551} C_VEL
LIN {X 0,Y 432.335,Z 330.255,A -85,B 0,C 180,E1 -9485.817,E2 -9485.817} C_VEL
LIN {X 0,Y 432.341,Z 330.249,A -85,B 0,C 180,E1 -9489.342,E2 -9489.342} C_VEL
LIN {X 0,Y 432.327,Z 330.251,A -85,B 0,C 180,E1 -9491.796,E2 -9491.796} C_VEL
LIN {X 0,Y 432.327,Z 330.256,A -85,B 0,C 180,E1 -9494.347,E2 -9494.347} C_VEL
LIN {X 0,Y 432.313,Z 330.253,A -85,B 0,C 180,E1 -9497.015,E2 -9497.015} C_VEL
LIN {X 0,Y 432.329,Z 330.256,A -85,B 0,C 180,E1 -9499.82,E2 -9499.82} C_VEL
LIN {X 0,Y 432.298,Z 330.258,A -85,B 0,C 180,E1 -9503.021,E2 -9503.021} C_VEL
LIN {X 0,Y 432.351,Z 330.254,A -85,B 0,C 180,E1 -9505.996,E2 -9505.996} C_VEL
LIN {X 0,Y 432.336,Z 330.243,A -85,B 0,C 180,E1 -9509.49,E2 -9509.49} C_VEL
LIN {X 0,Y 432.336,Z 330.249,A -85,B 0,C 180,E1 -9511.874,E2 -9511.874} C_VEL
LIN {X 0,Y 432.367,Z 330.249,A -85,B 0,C 180,E1 -9515.538,E2 -9515.538} C_VEL
LIN {X 0,Y 432.338,Z 330.251,A -85,B 0,C 180,E1 -9519.046,E2 -9519.046} C_VEL
LIN {X 0,Y 432.347,Z 330.255,A -85,B 0,C 180,E1 -9522.01,E2 -9522.01} C_VEL
LIN {X 0,Y 432.38,Z 330.246,A -85,B 0,C 180,E1 -9524.926,E2 -9524.926} C_VEL
LIN {X 0,Y 432.441,Z 330.238,A -85,B 0,C 180,E1 -9527.803,E2 -9527.803} C_VEL
LIN {X 0,Y 432.432,Z 330.244,A -85,B 0,C 180,E1 -9531.589,E2 -9531.589} C_VEL
LIN {X 0,Y 432.562,Z 330.224,A -85,B 0,C 180,E1 -9534.406,E2 -9534.406} C_VEL
LIN {X 0,Y 432.582,Z 330.219,A -85,B 0,C 180,E1 -9538.138,E2 -9538.138} C_VEL
LIN {X 0,Y 432.588,Z 330.223,A -85,B 0,C 180,E1 -9540,E2 -9540} C_VEL
LIN {X 0,Y 432.568,Z 330.221,A -85,B 0,C 180,E1 -9542.794,E2 -9542.794} C_VEL
LIN {X 0,Y 432.572,Z 330.226,A -85,B 0,C 180,E1 -9545.595,E2 -9545.595} C_VEL
LIN {X 0,Y 432.452,Z 330.236,A -85,B 0,C 180,E1 -9548.411,E2 -9548.411} C_VEL
LIN {X 0,Y 432.447,Z 330.233,A -85,B 0,C 180,E1 -9552.197,E2 -9552.197} C_VEL
LIN {X 0,Y 432.419,Z 330.239,A -85,B 0,C 180,E1 -9556.04,E2 -9556.04} C_VEL
LIN {X 0,Y 432.377,Z 330.248,A -85,B 0,C 180,E1 -9559.486,E2 -9559.486} C_VEL
LIN {X 0,Y 432.31,Z 330.262,A -85,B 0,C 180,E1 -9562.965,E2 -9562.965} C_VEL
LIN {X 0,Y 432.356,Z 330.251,A -85,B 0,C 180,E1 -9566.033,E2 -9566.033} C_VEL
LIN {X 0,Y 432.335,Z 330.256,A -85,B 0,C 180,E1 -9569.189,E2 -9569.189} C_VEL
LIN {X 0,Y 432.316,Z 330.257,A -85,B 0,C 180,E1 -9572.444,E2 -9572.444} C_VEL
LIN {X 0,Y 432.338,Z 330.252,A -85,B 0,C 180,E1 -9575.633,E2 -9575.633} C_VEL
LIN {X 0,Y 432.333,Z 330.258,A -85,B 0,C 180,E1 -9578.715,E2 -9578.715} C_VEL
LIN {X 0,Y 432.329,Z 330.255,A -85,B 0,C 180,E1 -9581.798,E2 -9581.798} C_VEL
LIN {X 0,Y 432.33,Z 330.259,A -85,B 0,C 180,E1 -9584.348,E2 -9584.348} C_VEL
LIN {X 0,Y 432.318,Z 330.259,A -85,B 0,C 180,E1 -9587.017,E2 -9587.017} C_VEL
LIN {X 0,Y 432.339,Z 330.257,A -85,B 0,C 180,E1 -9589.821,E2 -9589.821} C_VEL
LIN {X 0,Y 432.315,Z 330.258,A -85,B 0,C 180,E1 -9593.024,E2 -9593.024} C_VEL
LIN {X 0,Y 432.36,Z 330.253,A -85,B 0,C 180,E1 -9595.998,E2 -9595.998} C_VEL
LIN {X 0,Y 432.349,Z 330.452,A -85,B 0,C 180,E1 -9597.91,E2 -9597.91} C_VEL
LIN {X 0,Y 435.127,Z 342.635,A -85,B 0,C 180,E1 -9600.715,E2 -9600.715} C_VEL
LIN {X 0,Y 435.745,Z 346.236,A -85,B 0,C 180,E1 -9601.507,E2 -9601.507} C_VEL
LIN {X 0,Y 439.805,Z 362.829,A -85,B 0,C 180,E1 -9602.04,E2 -9602.04} C_VEL
LIN {X 0,Y 441.024,Z 368.969,A -85,B 0,C 180,E1 -9602.218,E2 -9602.218} C_VEL
LIN {X 0,Y 439.313,Z 483.346,A -85,B 0,C 180,E1 -9604.14,E2 -9604.14} C_VEL
LIN {X 0,Y 438.831,Z 497.623,A -85,B 0,C 180,E1 -9604.571,E2 -9604.571} C_VEL
LIN {X 0,Y 438.246,Z 511.182,A -85,B 0,C 180,E1 -9605.169,E2 -9605.169} C_VEL
LIN {X 0,Y 437.409,Z 524.394,A -85,B 0,C 180,E1 -9605.94,E2 -9605.94} C_VEL
LIN {X 0,Y 436.46,Z 537.173,A -85,B 0,C 180,E1 -9606.894,E2 -9606.894} C_VEL
LIN {X 0,Y 435.558,Z 548.714,A -85,B 0,C 180,E1 -9607.967,E2 -9607.967} C_VEL
LIN {X 0,Y 434.826,Z 557.324,A -85,B 0,C 180,E1 -9608.924,E2 -9608.924} C_VEL
LIN {X 0,Y 434.713,Z 559.336,A -85,B 0,C 180,E1 -9609.17,E2 -9609.17} C_VEL
LIN {X 0,Y 433.707,Z 563.62,A -85,B 0,C 180,E1 -9609.696,E2 -9609.696} C_VEL
LIN {X 0,Y 430.292,Z 570.346,A -85,B 0,C 180,E1 -9610.551,E2 -9610.551} C_VEL
LIN {X 0,Y 426.918,Z 576.585,A -85,B 0,C 180,E1 -9611.475,E2 -9611.475} C_VEL
LIN {X 0,Y 425.988,Z 580.067,A -85,B 0,C 180,E1 -9612.102,E2 -9612.102} C_VEL
LIN {X 0,Y 425.35,Z 587.467,A -85,B 0,C 180,E1 -9613.687,E2 -9613.687} C_VEL
LIN {X 0,Y 424.883,Z 593.062,A -85,B 0,C 180,E1 -9615.145,E2 -9615.145} C_VEL
LIN {X 0,Y 424.511,Z 598.897,A -85,B 0,C 180,E1 -9617.086,E2 -9617.086} C_VEL
LIN {X 0,Y 424.316,Z 602.239,A -85,B 0,C 180,E1 -9618.536,E2 -9618.536} C_VEL
LIN {X 0,Y 424.078,Z 605.344,A -85,B 0,C 180,E1 -9620.461,E2 -9620.461} C_VEL
LIN {X 0,Y 424.089,Z 607.061,A -85,B 0,C 180,E1 -9622.382,E2 -9622.382} C_VEL
LIN {X 0,Y 424.129,Z 607.444,A -85,B 0,C 180,E1 -9624.294,E2 -9624.294} C_VEL
LIN {X 0,Y 424.098,Z 606.509,A -85,B 0,C 180,E1 -9626.199,E2 -9626.199} C_VEL
LIN {X 0,Y 424.18,Z 604.243,A -85,B 0,C 180,E1 -9628.101,E2 -9628.101} C_VEL
LIN {X 0,Y 424.282,Z 600.601,A -85,B 0,C 180,E1 -9630,E2 -9630} C_VEL
LIN {X 0,Y 424.495,Z 595.477,A -85,B 0,C 180,E1 -9631.897,E2 -9631.897} C_VEL
LIN {X 0,Y 424.843,Z 590.502,A -85,B 0,C 180,E1 -9633.319,E2 -9633.319} C_VEL
LIN {X 0,Y 425.355,Z 583.407,A -85,B 0,C 180,E1 -9634.976,E2 -9634.976} C_VEL
LIN {X 0,Y 426.029,Z 575.982,A -85,B 0,C 180,E1 -9636.393,E2 -9636.393} C_VEL
LIN {X 0,Y 426.778,Z 567.083,A -85,B 0,C 180,E1 -9637.808,E2 -9637.808} C_VEL
LIN {X 0,Y 427.653,Z 556.414,A -85,B 0,C 180,E1 -9639.209,E2 -9639.209} C_VEL
LIN {X 0,Y 428.473,Z 545.42,A -85,B 0,C 180,E1 -9640.394,E2 -9640.394} C_VEL
LIN {X 0,Y 429.353,Z 533.448,A -85,B 0,C 180,E1 -9641.447,E2 -9641.447} C_VEL
LIN {X 0,Y 430.1,Z 521.951,A -85,B 0,C 180,E1 -9642.264,E2 -9642.264} C_VEL
LIN {X 0,Y 430.888,Z 508.391,A -85,B 0,C 180,E1 -9643.019,E2 -9643.019} C_VEL
LIN {X 0,Y 431.463,Z 494.971,A -85,B 0,C 180,E1 -9643.571,E2 -9643.571} C_VEL
LIN {X 0,Y 431.821,Z 481.504,A -85,B 0,C 180,E1 -9643.95,E2 -9643.95} C_VEL
LIN {X 0,Y 433.18,Z 369.002,A -85,B 0,C 180,E1 -9645.846,E2 -9645.846} C_VEL
LIN {X 0,Y 428.324,Z 346.205,A -85,B 0,C 180,E1 -9646.497,E2 -9646.497} C_VEL
LIN {X 0,Y 426.374,Z 335.923,A -85,B 0,C 180,E1 -9648.748,E2 -9648.748} C_VEL
LIN {X 0,Y 425.307,Z 331.137,A -85,B 0,C 180,E1 -9649.857,E2 -9649.857} C_VEL
LIN {X 0,Y 425.308,Z 331.132,A -85,B 0,C 180,E1 -9653.364,E2 -9653.364} C_VEL
LIN {X 0,Y 425.349,Z 331.125,A -85,B 0,C 180,E1 -9656.843,E2 -9656.843} C_VEL
LIN {X 0,Y 425.292,Z 331.134,A -85,B 0,C 180,E1 -9659.718,E2 -9659.718} C_VEL
LIN {X 0,Y 425.283,Z 331.133,A -85,B 0,C 180,E1 -9663.047,E2 -9663.047} C_VEL
LIN {X 0,Y 425.284,Z 331.131,A -85,B 0,C 180,E1 -9665.928,E2 -9665.928} C_VEL
LIN {X 0,Y 425.299,Z 331.131,A -85,B 0,C 180,E1 -9669.043,E2 -9669.043} C_VEL
LIN {X 0,Y 425.272,Z 331.133,A -85,B 0,C 180,E1 -9672.652,E2 -9672.652} C_VEL
LIN {X 0,Y 425.258,Z 331.136,A -85,B 0,C 180,E1 -9676.043,E2 -9676.043} C_VEL
LIN {X 0,Y 425.269,Z 331.13,A -85,B 0,C 180,E1 -9678.62,E2 -9678.62} C_VEL
LIN {X 0,Y 425.293,Z 331.135,A -85,B 0,C 180,E1 -9681.1,E2 -9681.1} C_VEL
LIN {X 0,Y 425.292,Z 331.132,A -85,B 0,C 180,E1 -9684.663,E2 -9684.663} C_VEL
LIN {X 0,Y 425.256,Z 331.134,A -85,B 0,C 180,E1 -9688.072,E2 -9688.072} C_VEL
LIN {X 0,Y 425.323,Z 331.122,A -85,B 0,C 180,E1 -9691.367,E2 -9691.367} C_VEL
LIN {X 0,Y 425.273,Z 331.131,A -85,B 0,C 180,E1 -9694.553,E2 -9694.553} C_VEL
LIN {X 0,Y 425.274,Z 331.136,A -85,B 0,C 180,E1 -9696.632,E2 -9696.632} C_VEL
LIN {X 0,Y 425.285,Z 331.12,A -85,B 0,C 180,E1 -9699.694,E2 -9699.694} C_VEL
LIN {X 0,Y 425.322,Z 331.129,A -85,B 0,C 180,E1 -9702.696,E2 -9702.696} C_VEL
LIN {X 0,Y 425.334,Z 331.12,A -85,B 0,C 180,E1 -9705.649,E2 -9705.649} C_VEL
LIN {X 0,Y 425.335,Z 331.118,A -85,B 0,C 180,E1 -9708.563,E2 -9708.563} C_VEL
LIN {X 0,Y 425.494,Z 331.108,A -85,B 0,C 180,E1 -9712.31,E2 -9712.31} C_VEL
LIN {X 0,Y 425.527,Z 331.099,A -85,B 0,C 180,E1 -9714.313,E2 -9714.313} C_VEL
LIN {X 0,Y 425.555,Z 331.096,A -85,B 0,C 180,E1 -9718.107,E2 -9718.107} C_VEL
LIN {X 0,Y 425.495,Z 331.105,A -85,B 0,C 180,E1 -9720.946,E2 -9720.946} C_VEL
LIN {X 0,Y 425.496,Z 331.1,A -85,B 0,C 180,E1 -9722.84,E2 -9722.84} C_VEL
LIN {X 0,Y 425.497,Z 331.105,A -85,B 0,C 180,E1 -9725.687,E2 -9725.687} C_VEL
LIN {X 0,Y 425.385,Z 331.116,A -85,B 0,C 180,E1 -9728.551,E2 -9728.551} C_VEL
LIN {X 0,Y 425.399,Z 331.123,A -85,B 0,C 180,E1 -9732.402,E2 -9732.402} C_VEL
LIN {X 0,Y 425.376,Z 331.119,A -85,B 0,C 180,E1 -9736.312,E2 -9736.312} C_VEL
LIN {X 0,Y 425.317,Z 331.128,A -85,B 0,C 180,E1 -9739.636,E2 -9739.636} C_VEL
LIN {X 0,Y 425.277,Z 331.135,A -85,B 0,C 180,E1 -9742.339,E2 -9742.339} C_VEL
LIN {X 0,Y 425.309,Z 331.127,A -85,B 0,C 180,E1 -9744.657,E2 -9744.657} C_VEL
LIN {X 0,Y 425.261,Z 331.133,A -85,B 0,C 180,E1 -9747.564,E2 -9747.564} C_VEL
LIN {X 0,Y 425.281,Z 331.129,A -85,B 0,C 180,E1 -9750.761,E2 -9750.761} C_VEL
LIN {X 0,Y 425.303,Z 331.131,A -85,B 0,C 180,E1 -9754.289,E2 -9754.289} C_VEL
LIN {X 0,Y 425.272,Z 331.136,A -85,B 0,C 180,E1 -9757.695,E2 -9757.695} C_VEL
LIN {X 0,Y 425.276,Z 331.128,A -85,B 0,C 180,E1 -9760.522,E2 -9760.522} C_VEL
LIN {X 0,Y 425.251,Z 331.137,A -85,B 0,C 180,E1 -9763.352,E2 -9763.352} C_VEL
LIN {X 0,Y 425.251,Z 331.136,A -85,B 0,C 180,E1 -9766.65,E2 -9766.65} C_VEL
LIN {X 0,Y 425.28,Z 331.138,A -85,B 0,C 180,E1 -9769.873,E2 -9769.873} C_VEL
LIN {X 0,Y 425.273,Z 331.137,A -85,B 0,C 180,E1 -9772.489,E2 -9772.489} C_VEL
LIN {X 0,Y 425.304,Z 331.135,A -85,B 0,C 180,E1 -9775.818,E2 -9775.818} C_VEL
LIN {X 0,Y 425.287,Z 331.137,A -85,B 0,C 180,E1 -9779.24,E2 -9779.24} C_VEL
LIN {X 0,Y 425.327,Z 331.214,A -85,B 0,C 180,E1 -9780.641,E2 -9780.641} C_VEL
LIN {X 0,Y 428.131,Z 343.892,A -85,B 0,C 180,E1 -9783.166,E2 -9783.166} C_VEL
LIN {X 0,Y 429.35,Z 350.256,A -85,B 0,C 180,E1 -9784.392,E2 -9784.392} C_VEL
LIN {X 0,Y 428.206,Z 368.049,A -85,B 0,C 180,E1 -9787.53,E2 -9787.53} C_VEL
LIN {X 0,Y 433.041,Z 396.739,A -85,B 0,C 180,E1 -9788.267,E2 -9788.267} C_VEL
LIN {X 0,Y 431.558,Z 505.624,A -85,B 0,C 180,E1 -9790.096,E2 -9790.096} C_VEL
LIN {X 0,Y 431.079,Z 519.75,A -85,B 0,C 180,E1 -9790.507,E2 -9790.507} C_VEL
LIN {X 0,Y 430.431,Z 532.347,A -85,B 0,C 180,E1 -9791.034,E2 -9791.034} C_VEL
LIN {X 0,Y 429.699,Z 545.507,A -85,B 0,C 180,E1 -9791.774,E2 -9791.774} C_VEL
LIN {X 0,Y 428.773,Z 558.581,A -85,B 0,C 180,E1 -9792.718,E2 -9792.718} C_VEL
LIN {X 0,Y 427.771,Z 570.443,A -85,B 0,C 180,E1 -9793.782,E2 -9793.782} C_VEL
LIN {X 0,Y 426.913,Z 581.293,A -85,B 0,C 180,E1 -9794.973,E2 -9794.973} C_VEL
LIN {X 0,Y 426.151,Z 592.03,A -85,B 0,C 180,E1 -9796.408,E2 -9796.408} C_VEL
LIN {X 0,Y 425.486,Z 600.882,A -85,B 0,C 180,E1 -9797.843,E2 -9797.843} C_VEL
LIN {X 0,Y 424.988,Z 608.238,A -85,B 0,C 180,E1 -9799.279,E2 -9799.279} C_VEL
LIN {X 0,Y 424.556,Z 615.273,A -85,B 0,C 180,E1 -9800.952,E2 -9800.952} C_VEL
LIN {X 0,Y 424.324,Z 621.586,A -85,B 0,C 180,E1 -9802.864,E2 -9802.864} C_VEL
LIN {X 0,Y 424.192,Z 625.178,A -85,B 0,C 180,E1 -9804.295,E2 -9804.295} C_VEL
LIN {X 0,Y 424.088,Z 628.693,A -85,B 0,C 180,E1 -9806.199,E2 -9806.199} C_VEL
LIN {X 0,Y 424.126,Z 630.805,A -85,B 0,C 180,E1 -9808.101,E2 -9808.101} C_VEL
LIN {X 0,Y 424.082,Z 631.562,A -85,B 0,C 180,E1 -9810,E2 -9810} C_VEL
LIN {X 0,Y 424.126,Z 630.988,A -85,B 0,C 180,E1 -9811.899,E2 -9811.899} C_VEL
LIN {X 0,Y 424.087,Z 629.068,A -85,B 0,C 180,E1 -9813.801,E2 -9813.801} C_VEL
LIN {X 0,Y 424.193,Z 625.751,A -85,B 0,C 180,E1 -9815.705,E2 -9815.705} C_VEL
LIN {X 0,Y 424.316,Z 622.289,A -85,B 0,C 180,E1 -9817.136,E2 -9817.136} C_VEL
LIN {X 0,Y 424.594,Z 616.316,A -85,B 0,C 180,E1 -9819.047,E2 -9819.047} C_VEL
LIN {X 0,Y 425.041,Z 609.604,A -85,B 0,C 180,E1 -9820.72,E2 -9820.72} C_VEL
LIN {X 0,Y 425.732,Z 601.267,A -85,B 0,C 180,E1 -9822.392,E2 -9822.392} C_VEL
LIN {X 0,Y 426.393,Z 592.596,A -85,B 0,C 180,E1 -9823.827,E2 -9823.827} C_VEL
LIN {X 0,Y 427.303,Z 582.107,A -85,B 0,C 180,E1 -9825.257,E2 -9825.257} C_VEL
LIN {X 0,Y 428.38,Z 570.391,A -85,B 0,C 180,E1 -9826.562,E2 -9826.562} C_VEL
LIN {X 0,Y 429.408,Z 558.672,A -85,B 0,C 180,E1 -9827.624,E2 -9827.624} C_VEL
LIN {X 0,Y 430.309,Z 547.094,A -85,B 0,C 180,E1 -9828.478,E2 -9828.478} C_VEL
LIN {X 0,Y 431.185,Z 533.463,A -85,B 0,C 180,E1 -9829.272,E2 -9829.272} C_VEL
LIN {X 0,Y 431.916,Z 520.702,A -85,B 0,C 180,E1 -9829.825,E2 -9829.825} C_VEL
LIN {X 0,Y 432.522,Z 506.222,A -85,B 0,C 180,E1 -9830.261,E2 -9830.261} C_VEL
LIN {X 0,Y 434.173,Z 396.508,A -85,B 0,C 180,E1 -9832.132,E2 -9832.132} C_VEL
LIN {X 0,Y 430.484,Z 376.033,A -85,B 0,C 180,E1 -9832.716,E2 -9832.716} C_VEL
LIN {X 0,Y 428.768,Z 367.845,A -85,B 0,C 180,E1 -9832.978,E2 -9832.978} C_VEL
LIN {X 0,Y 429.976,Z 352.364,A -85,B 0,C 180,E1 -9835.77,E2 -9835.77} C_VEL
LIN {X 0,Y 427.855,Z 341.659,A -85,B 0,C 180,E1 -9837.939,E2 -9837.939} C_VEL
LIN {X 0,Y 425.298,Z 331.136,A -85,B 0,C 180,E1 -9840.196,E2 -9840.196} C_VEL
LIN {X 0,Y 425.279,Z 331.137,A -85,B 0,C 180,E1 -9843.047,E2 -9843.047} C_VEL
LIN {X 0,Y 425.279,Z 331.135,A -85,B 0,C 180,E1 -9845.928,E2 -9845.928} C_VEL
LIN {X 0,Y 425.288,Z 331.129,A -85,B 0,C 180,E1 -9849.042,E2 -9849.042} C_VEL
LIN {X 0,Y 425.268,Z 331.132,A -85,B 0,C 180,E1 -9852.652,E2 -9852.652} C_VEL
LIN {X 0,Y 425.255,Z 331.135,A -85,B 0,C 180,E1 -9856.043,E2 -9856.043} C_VEL
LIN {X 0,Y 425.267,Z 331.136,A -85,B 0,C 180,E1 -9858.621,E2 -9858.621} C_VEL
LIN {X 0,Y 425.299,Z 331.131,A -85,B 0,C 180,E1 -9861.102,E2 -9861.102} C_VEL
LIN {X 0,Y 425.291,Z 331.13,A -85,B 0,C 180,E1 -9864.663,E2 -9864.663} C_VEL
LIN {X 0,Y 425.255,Z 331.133,A -85,B 0,C 180,E1 -9868.072,E2 -9868.072} C_VEL
LIN {X 0,Y 425.303,Z 331.119,A -85,B 0,C 180,E1 -9871.366,E2 -9871.366} C_VEL
LIN {X 0,Y 425.26,Z 331.133,A -85,B 0,C 180,E1 -9874.553,E2 -9874.553} C_VEL
LIN {X 0,Y 425.273,Z 331.133,A -85,B 0,C 180,E1 -9876.633,E2 -9876.633} C_VEL
LIN {X 0,Y 425.284,Z 331.131,A -85,B 0,C 180,E1 -9879.694,E2 -9879.694} C_VEL
LIN {X 0,Y 425.321,Z 331.126,A -85,B 0,C 180,E1 -9882.697,E2 -9882.697} C_VEL
LIN {X 0,Y 425.333,Z 331.131,A -85,B 0,C 180,E1 -9885.65,E2 -9885.65} C_VEL
LIN {X 0,Y 425.319,Z 331.122,A -85,B 0,C 180,E1 -9888.563,E2 -9888.563} C_VEL
LIN {X 0,Y 425.381,Z 331.124,A -85,B 0,C 180,E1 -9891.449,E2 -9891.449} C_VEL
LIN {X 0,Y 425.516,Z 331.102,A -85,B 0,C 180,E1 -9894.313,E2 -9894.313} C_VEL
LIN {X 0,Y 425.551,Z 331.094,A -85,B 0,C 180,E1 -9898.107,E2 -9898.107} C_VEL
LIN {X 0,Y 425.425,Z 331.117,A -85,B 0,C 180,E1 -9900.947,E2 -9900.947} C_VEL
LIN {X 0,Y 425.522,Z 331.099,A -85,B 0,C 180,E1 -9902.84,E2 -9902.84} C_VEL
LIN {X 0,Y 425.492,Z 331.105,A -85,B 0,C 180,E1 -9906.596,E2 -9906.596} C_VEL
LIN {X 0,Y 425.384,Z 331.123,A -85,B 0,C 180,E1 -9909.51,E2 -9909.51} C_VEL
LIN {X 0,Y 425.383,Z 331.117,A -85,B 0,C 180,E1 -9912.904,E2 -9912.904} C_VEL
LIN {X 0,Y 425.351,Z 331.122,A -85,B 0,C 180,E1 -9916.605,E2 -9916.605} C_VEL
LIN {X 0,Y 425.319,Z 331.126,A -85,B 0,C 180,E1 -9919.636,E2 -9919.636} C_VEL
LIN {X 0,Y 425.279,Z 331.133,A -85,B 0,C 180,E1 -9922.34,E2 -9922.34} C_VEL
LIN {X 0,Y 425.287,Z 331.133,A -85,B 0,C 180,E1 -9925.446,E2 -9925.446} C_VEL
LIN {X 0,Y 425.323,Z 331.128,A -85,B 0,C 180,E1 -9928.633,E2 -9928.633} C_VEL
LIN {X 0,Y 425.258,Z 331.132,A -85,B 0,C 180,E1 -9931.928,E2 -9931.928} C_VEL
LIN {X 0,Y 425.293,Z 331.131,A -85,B 0,C 180,E1 -9935.337,E2 -9935.337} C_VEL
LIN {X 0,Y 425.292,Z 331.133,A -85,B 0,C 180,E1 -9938.9,E2 -9938.9} C_VEL
LIN {X 0,Y 425.286,Z 331.134,A -85,B 0,C 180,E1 -9941.959,E2 -9941.959} C_VEL
LIN {X 0,Y 425.282,Z 331.134,A -85,B 0,C 180,E1 -9945.284,E2 -9945.284} C_VEL
LIN {X 0,Y 425.273,Z 331.137,A -85,B 0,C 180,E1 -9948.623,E2 -9948.623} C_VEL
LIN {X 0,Y 425.314,Z 331.131,A -85,B 0,C 180,E1 -9951.104,E2 -9951.104} C_VEL
LIN {X 0,Y 425.3,Z 331.129,A -85,B 0,C 180,E1 -9954.665,E2 -9954.665} C_VEL
LIN {X 0,Y 425.3,Z 331.209,A -85,B 0,C 180,E1 -9957.525,E2 -9957.525} C_VEL
LIN {X 0,Y 428.143,Z 343.713,A -85,B 0,C 180,E1 -9960.46,E2 -9960.46} C_VEL
LIN {X 0,Y 428.756,Z 346.674,A -85,B 0,C 180,E1 -9961.087,E2 -9961.087} C_VEL
LIN {X 0,Y 431.438,Z 355.791,A -85,B 0,C 180,E1 -9961.417,E2 -9961.417} C_VEL
LIN {X 0,Y 434.486,Z 369.439,A -85,B 0,C 180,E1 -9961.845,E2 -9961.845} C_VEL
LIN {X 0,Y 432.751,Z 482.752,A -85,B 0,C 180,E1 -9963.773,E2 -9963.773} C_VEL
LIN {X 0,Y 432.246,Z 497.554,A -85,B 0,C 180,E1 -9964.22,E2 -9964.22} C_VEL
LIN {X 0,Y 431.619,Z 511.178,A -85,B 0,C 180,E1 -9964.825,E2 -9964.825} C_VEL
LIN {X 0,Y 430.83,Z 523.537,A -85,B 0,C 180,E1 -9965.548,E2 -9965.548} C_VEL
LIN {X 0,Y 429.895,Z 535.909,A -85,B 0,C 180,E1 -9966.466,E2 -9966.466} C_VEL
LIN {X 0,Y 428.959,Z 547.017,A -85,B 0,C 180,E1 -9967.483,E2 -9967.483} C_VEL
LIN {X 0,Y 428.028,Z 556.933,A -85,B 0,C 180,E1 -9968.572,E2 -9968.572} C_VEL
LIN {X 0,Y 427.278,Z 566.204,A -85,B 0,C 180,E1 -9969.794,E2 -9969.794} C_VEL
LIN {X 0,Y 426.405,Z 575.449,A -85,B 0,C 180,E1 -9971.253,E2 -9971.253} C_VEL
LIN {X 0,Y 425.988,Z 580.067,A -85,B 0,C 180,E1 -9972.102,E2 -9972.102} C_VEL
LIN {X 0,Y 425.079,Z 583.408,A -85,B 0,C 180,E1 -9972.751,E2 -9972.751} C_VEL
LIN {X 0,Y 421.805,Z 588.511,A -85,B 0,C 180,E1 -9973.815,E2 -9973.815} C_VEL
LIN {X 0,Y 418.555,Z 593.085,A -85,B 0,C 180,E1 -9974.933,E2 -9974.933} C_VEL
LIN {X 0,Y 417.698,Z 595.505,A -85,B 0,C 180,E1 -9975.661,E2 -9975.661} C_VEL
LIN {X 0,Y 417.372,Z 600.698,A -85,B 0,C 180,E1 -9977.595,E2 -9977.595} C_VEL
LIN {X 0,Y 417.114,Z 604.063,A -85,B 0,C 180,E1 -9979.319,E2 -9979.319} C_VEL
LIN {X 0,Y 416.989,Z 606.514,A -85,B 0,C 180,E1 -9981.276,E2 -9981.276} C_VEL
LIN {X 0,Y 417.029,Z 607.607,A -85,B 0,C 180,E1 -9983.225,E2 -9983.225} C_VEL
LIN {X 0,Y 417.041,Z 607.378,A -85,B 0,C 180,E1 -9985.167,E2 -9985.167} C_VEL
LIN {X 0,Y 417.072,Z 605.828,A -85,B 0,C 180,E1 -9987.102,E2 -9987.102} C_VEL
LIN {X 0,Y 417.113,Z 602.935,A -85,B 0,C 180,E1 -9989.035,E2 -9989.035} C_VEL
LIN {X 0,Y 417.303,Z 598.618,A -85,B 0,C 180,E1 -9990.965,E2 -9990.965} C_VEL
LIN {X 0,Y 417.625,Z 592.75,A -85,B 0,C 180,E1 -9992.894,E2 -9992.894} C_VEL
LIN {X 0,Y 418.197,Z 586.136,A -85,B 0,C 180,E1 -9994.578,E2 -9994.578} C_VEL
LIN {X 0,Y 418.864,Z 577.924,A -85,B 0,C 180,E1 -9996.261,E2 -9996.261} C_VEL
LIN {X 0,Y 419.696,Z 569.366,A -85,B 0,C 180,E1 -9997.698,E2 -9997.698} C_VEL
LIN {X 0,Y 420.475,Z 559.233,A -85,B 0,C 180,E1 -9999.11,E2 -9999.11} C_VEL
LIN {X 0,Y 421.346,Z 548.628,A -85,B 0,C 180,E1 -10000.329,E2 -10000.329} C_VEL
LIN {X 0,Y 422.279,Z 537.3,A -85,B 0,C 180,E1 -10001.398,E2 -10001.398} C_VEL
LIN {X 0,Y 423.129,Z 524.917,A -85,B 0,C 180,E1 -10002.348,E2 -10002.348} C_VEL
LIN {X 0,Y 423.91,Z 512.188,A -85,B 0,C 180,E1 -10003.116,E2 -10003.116} C_VEL
LIN {X 0,Y 424.553,Z 498.587,A -85,B 0,C 180,E1 -10003.735,E2 -10003.735} C_VEL
LIN {X 0,Y 425.031,Z 484.572,A -85,B 0,C 180,E1 -10004.177,E2 -10004.177} C_VEL
LIN {X 0,Y 425.469,Z 455.124,A -85,B 0,C 180,E1 -10004.712,E2 -10004.712} C_VEL
LIN {X 0,Y 426.483,Z 369.765,A -85,B 0,C 180,E1 -10006.163,E2 -10006.163} C_VEL
LIN {X 0,Y 421.799,Z 348.258,A -85,B 0,C 180,E1 -10006.784,E2 -10006.784} C_VEL
LIN {X 0,Y 421.251,Z 346.427,A -85,B 0,C 180,E1 -10006.856,E2 -10006.856} C_VEL
LIN {X 0,Y 418.977,Z 335.316,A -85,B 0,C 180,E1 -10009.347,E2 -10009.347} C_VEL
LIN {X 0,Y 418.273,Z 332.013,A -85,B 0,C 180,E1 -10010.114,E2 -10010.114} C_VEL
LIN {X 0,Y 418.288,Z 332.009,A -85,B 0,C 180,E1 -10013.78,E2 -10013.78} C_VEL
LIN {X 0,Y 418.312,Z 332.003,A -85,B 0,C 180,E1 -10017.07,E2 -10017.07} C_VEL
LIN {X 0,Y 418.246,Z 332.011,A -85,B 0,C 180,E1 -10020.271,E2 -10020.271} C_VEL
LIN {X 0,Y 418.249,Z 332.014,A -85,B 0,C 180,E1 -10023.676,E2 -10023.676} C_VEL
LIN {X 0,Y 418.245,Z 332.01,A -85,B 0,C 180,E1 -10027.222,E2 -10027.222} C_VEL
LIN {X 0,Y 418.25,Z 332.001,A -85,B 0,C 180,E1 -10029.681,E2 -10029.681} C_VEL
LIN {X 0,Y 418.227,Z 332.01,A -85,B 0,C 180,E1 -10032.32,E2 -10032.32} C_VEL
LIN {X 0,Y 418.232,Z 332.011,A -85,B 0,C 180,E1 -10035.107,E2 -10035.107} C_VEL
LIN {X 0,Y 418.236,Z 332.008,A -85,B 0,C 180,E1 -10037.766,E2 -10037.766} C_VEL
LIN {X 0,Y 418.241,Z 332.01,A -85,B 0,C 180,E1 -10040.619,E2 -10040.619} C_VEL
LIN {X 0,Y 418.236,Z 332.01,A -85,B 0,C 180,E1 -10043.975,E2 -10043.975} C_VEL
LIN {X 0,Y 418.25,Z 332.008,A -85,B 0,C 180,E1 -10047.155,E2 -10047.155} C_VEL
LIN {X 0,Y 418.261,Z 332.009,A -85,B 0,C 180,E1 -10050.894,E2 -10050.894} C_VEL
LIN {X 0,Y 418.252,Z 332.004,A -85,B 0,C 180,E1 -10054.094,E2 -10054.094} C_VEL
LIN {X 0,Y 418.222,Z 332.011,A -85,B 0,C 180,E1 -10057.262,E2 -10057.262} C_VEL
LIN {X 0,Y 418.273,Z 331.994,A -85,B 0,C 180,E1 -10060.363,E2 -10060.363} C_VEL
LIN {X 0,Y 418.306,Z 332.002,A -85,B 0,C 180,E1 -10063.404,E2 -10063.404} C_VEL
LIN {X 0,Y 418.335,Z 331.987,A -85,B 0,C 180,E1 -10066.999,E2 -10066.999} C_VEL
LIN {X 0,Y 418.324,Z 331.998,A -85,B 0,C 180,E1 -10070.328,E2 -10070.328} C_VEL
LIN {X 0,Y 418.455,Z 331.978,A -85,B 0,C 180,E1 -10073.248,E2 -10073.248} C_VEL
LIN {X 0,Y 418.313,Z 331.986,A -85,B 0,C 180,E1 -10075.181,E2 -10075.181} C_VEL
LIN {X 0,Y 418.524,Z 331.971,A -85,B 0,C 180,E1 -10078.075,E2 -10078.075} C_VEL
LIN {X 0,Y 418.458,Z 331.981,A -85,B 0,C 180,E1 -10080.962,E2 -10080.962} C_VEL
LIN {X 0,Y 418.453,Z 331.977,A -85,B 0,C 180,E1 -10082.888,E2 -10082.888} C_VEL
LIN {X 0,Y 418.457,Z 331.982,A -85,B 0,C 180,E1 -10085.783,E2 -10085.783} C_VEL
LIN {X 0,Y 418.357,Z 331.989,A -85,B 0,C 180,E1 -10088.696,E2 -10088.696} C_VEL
LIN {X 0,Y 418.299,Z 332.001,A -85,B 0,C 180,E1 -10091.631,E2 -10091.631} C_VEL
LIN {X 0,Y 418.289,Z 332,A -85,B 0,C 180,E1 -10094.597,E2 -10094.597} C_VEL
LIN {X 0,Y 418.267,Z 332.004,A -85,B 0,C 180,E1 -10097.604,E2 -10097.604} C_VEL
LIN {X 0,Y 418.238,Z 332.002,A -85,B 0,C 180,E1 -10100.663,E2 -10100.663} C_VEL
LIN {X 0,Y 418.263,Z 332.008,A -85,B 0,C 180,E1 -10103.782,E2 -10103.782} C_VEL
LIN {X 0,Y 418.216,Z 332.009,A -85,B 0,C 180,E1 -10107.048,E2 -10107.048} C_VEL
LIN {X 0,Y 418.232,Z 332.01,A -85,B 0,C 180,E1 -10110.273,E2 -10110.273} C_VEL
LIN {X 0,Y 418.24,Z 332.013,A -85,B 0,C 180,E1 -10113.678,E2 -10113.678} C_VEL
LIN {X 0,Y 418.232,Z 332.01,A -85,B 0,C 180,E1 -10117.225,E2 -10117.225} C_VEL
LIN {X 0,Y 418.246,Z 332.012,A -85,B 0,C 180,E1 -10119.682,E2 -10119.682} C_VEL
LIN {X 0,Y 418.222,Z 332.011,A -85,B 0,C 180,E1 -10122.322,E2 -10122.322} C_VEL
LIN {X 0,Y 418.229,Z 332.011,A -85,B 0,C 180,E1 -10125.109,E2 -10125.109} C_VEL
LIN {X 0,Y 418.234,Z 332.016,A -85,B 0,C 180,E1 -10127.768,E2 -10127.768} C_VEL
LIN {X 0,Y 418.24,Z 332.013,A -85,B 0,C 180,E1 -10130.621,E2 -10130.621} C_VEL
LIN {X 0,Y 418.24,Z 332.016,A -85,B 0,C 180,E1 -10133.977,E2 -10133.977} C_VEL
LIN {X 0,Y 418.254,Z 332.014,A -85,B 0,C 180,E1 -10137.157,E2 -10137.157} C_VEL
LIN {X 0,Y 418.288,Z 332.187,A -85,B 0,C 180,E1 -10140.365,E2 -10140.365} C_VEL
LIN {X 0,Y 420.904,Z 343.898,A -85,B 0,C 180,E1 -10142.747,E2 -10142.747} C_VEL
LIN {X 0,Y 422.443,Z 352.187,A -85,B 0,C 180,E1 -10144.371,E2 -10144.371} C_VEL
LIN {X 0,Y 421.333,Z 367.857,A -85,B 0,C 180,E1 -10147.18,E2 -10147.18} C_VEL
LIN {X 0,Y 426.268,Z 396.477,A -85,B 0,C 180,E1 -10147.936,E2 -10147.936} C_VEL
LIN {X 0,Y 424.835,Z 505.408,A -85,B 0,C 180,E1 -10149.799,E2 -10149.799} C_VEL
LIN {X 0,Y 424.312,Z 519.539,A -85,B 0,C 180,E1 -10150.214,E2 -10150.214} C_VEL
LIN {X 0,Y 423.604,Z 533.025,A -85,B 0,C 180,E1 -10150.796,E2 -10150.796} C_VEL
LIN {X 0,Y 422.759,Z 546.61,A -85,B 0,C 180,E1 -10151.588,E2 -10151.588} C_VEL
LIN {X 0,Y 421.819,Z 559.457,A -85,B 0,C 180,E1 -10152.549,E2 -10152.549} C_VEL
LIN {X 0,Y 420.805,Z 571.133,A -85,B 0,C 180,E1 -10153.631,E2 -10153.631} C_VEL
LIN {X 0,Y 419.831,Z 582.818,A -85,B 0,C 180,E1 -10154.962,E2 -10154.962} C_VEL
LIN {X 0,Y 419.069,Z 593.267,A -85,B 0,C 180,E1 -10156.421,E2 -10156.421} C_VEL
LIN {X 0,Y 418.411,Z 601.88,A -85,B 0,C 180,E1 -10157.88,E2 -10157.88} C_VEL
LIN {X 0,Y 417.787,Z 610.098,A -85,B 0,C 180,E1 -10159.582,E2 -10159.582} C_VEL
LIN {X 0,Y 417.411,Z 616.718,A -85,B 0,C 180,E1 -10161.284,E2 -10161.284} C_VEL
LIN {X 0,Y 417.227,Z 622.588,A -85,B 0,C 180,E1 -10163.229,E2 -10163.229} C_VEL
LIN {X 0,Y 417.077,Z 626.865,A -85,B 0,C 180,E1 -10165.167,E2 -10165.167} C_VEL
LIN {X 0,Y 417.025,Z 629.687,A -85,B 0,C 180,E1 -10167.102,E2 -10167.102} C_VEL
LIN {X 0,Y 417.008,Z 631.136,A -85,B 0,C 180,E1 -10169.034,E2 -10169.034} C_VEL
LIN {X 0,Y 417.008,Z 631.244,A -85,B 0,C 180,E1 -10170.966,E2 -10170.966} C_VEL
LIN {X 0,Y 417.022,Z 630.021,A -85,B 0,C 180,E1 -10172.898,E2 -10172.898} C_VEL
LIN {X 0,Y 417.078,Z 627.438,A -85,B 0,C 180,E1 -10174.833,E2 -10174.833} C_VEL
LIN {X 0,Y 417.225,Z 623.41,A -85,B 0,C 180,E1 -10176.771,E2 -10176.771} C_VEL
LIN {X 0,Y 417.448,Z 617.833,A -85,B 0,C 180,E1 -10178.715,E2 -10178.715} C_VEL
LIN {X 0,Y 417.828,Z 611.555,A -85,B 0,C 180,E1 -10180.417,E2 -10180.417} C_VEL
LIN {X 0,Y 418.578,Z 603.754,A -85,B 0,C 180,E1 -10182.115,E2 -10182.115} C_VEL
LIN {X 0,Y 419.179,Z 595.624,A -85,B 0,C 180,E1 -10183.575,E2 -10183.575} C_VEL
LIN {X 0,Y 420.107,Z 585.846,A -85,B 0,C 180,E1 -10185.028,E2 -10185.028} C_VEL
LIN {X 0,Y 421.112,Z 575.008,A -85,B 0,C 180,E1 -10186.357,E2 -10186.357} C_VEL
LIN {X 0,Y 422.319,Z 563.013,A -85,B 0,C 180,E1 -10187.555,E2 -10187.555} C_VEL
LIN {X 0,Y 423.319,Z 551.114,A -85,B 0,C 180,E1 -10188.52,E2 -10188.52} C_VEL
LIN {X 0,Y 424.248,Z 538.301,A -85,B 0,C 180,E1 -10189.348,E2 -10189.348} C_VEL
LIN {X 0,Y 425.02,Z 525.067,A -85,B 0,C 180,E1 -10190.003,E2 -10190.003} C_VEL
LIN {X 0,Y 425.795,Z 510.59,A -85,B 0,C 180,E1 -10190.501,E2 -10190.501} C_VEL
LIN {X 0,Y 426.178,Z 495.26,A -85,B 0,C 180,E1 -10190.829,E2 -10190.829} C_VEL
LIN {X 0,Y 427.621,Z 397.014,A -85,B 0,C 180,E1 -10192.511,E2 -10192.511} C_VEL
LIN {X 0,Y 424.028,Z 377.185,A -85,B 0,C 180,E1 -10193.092,E2 -10193.092} C_VEL
LIN {X 0,Y 422.007,Z 367.665,A -85,B 0,C 180,E1 -10193.4,E2 -10193.4} C_VEL
LIN {X 0,Y 423.113,Z 353.518,A -85,B 0,C 180,E1 -10196.001,E2 -10196.001} C_VEL
LIN {X 0,Y 420.69,Z 341.82,A -85,B 0,C 180,E1 -10198.431,E2 -10198.431} C_VEL
LIN {X 0,Y 418.271,Z 332.011,A -85,B 0,C 180,E1 -10200.573,E2 -10200.573} C_VEL
LIN {X 0,Y 418.245,Z 332.013,A -85,B 0,C 180,E1 -10203.676,E2 -10203.676} C_VEL
LIN {X 0,Y 418.236,Z 332.002,A -85,B 0,C 180,E1 -10207.223,E2 -10207.223} C_VEL
LIN {X 0,Y 418.243,Z 332.005,A -85,B 0,C 180,E1 -10209.682,E2 -10209.682} C_VEL
LIN {X 0,Y 418.224,Z 332.013,A -85,B 0,C 180,E1 -10212.32,E2 -10212.32} C_VEL
LIN {X 0,Y 418.229,Z 332.005,A -85,B 0,C 180,E1 -10215.108,E2 -10215.108} C_VEL
LIN {X 0,Y 418.233,Z 332.009,A -85,B 0,C 180,E1 -10217.766,E2 -10217.766} C_VEL
